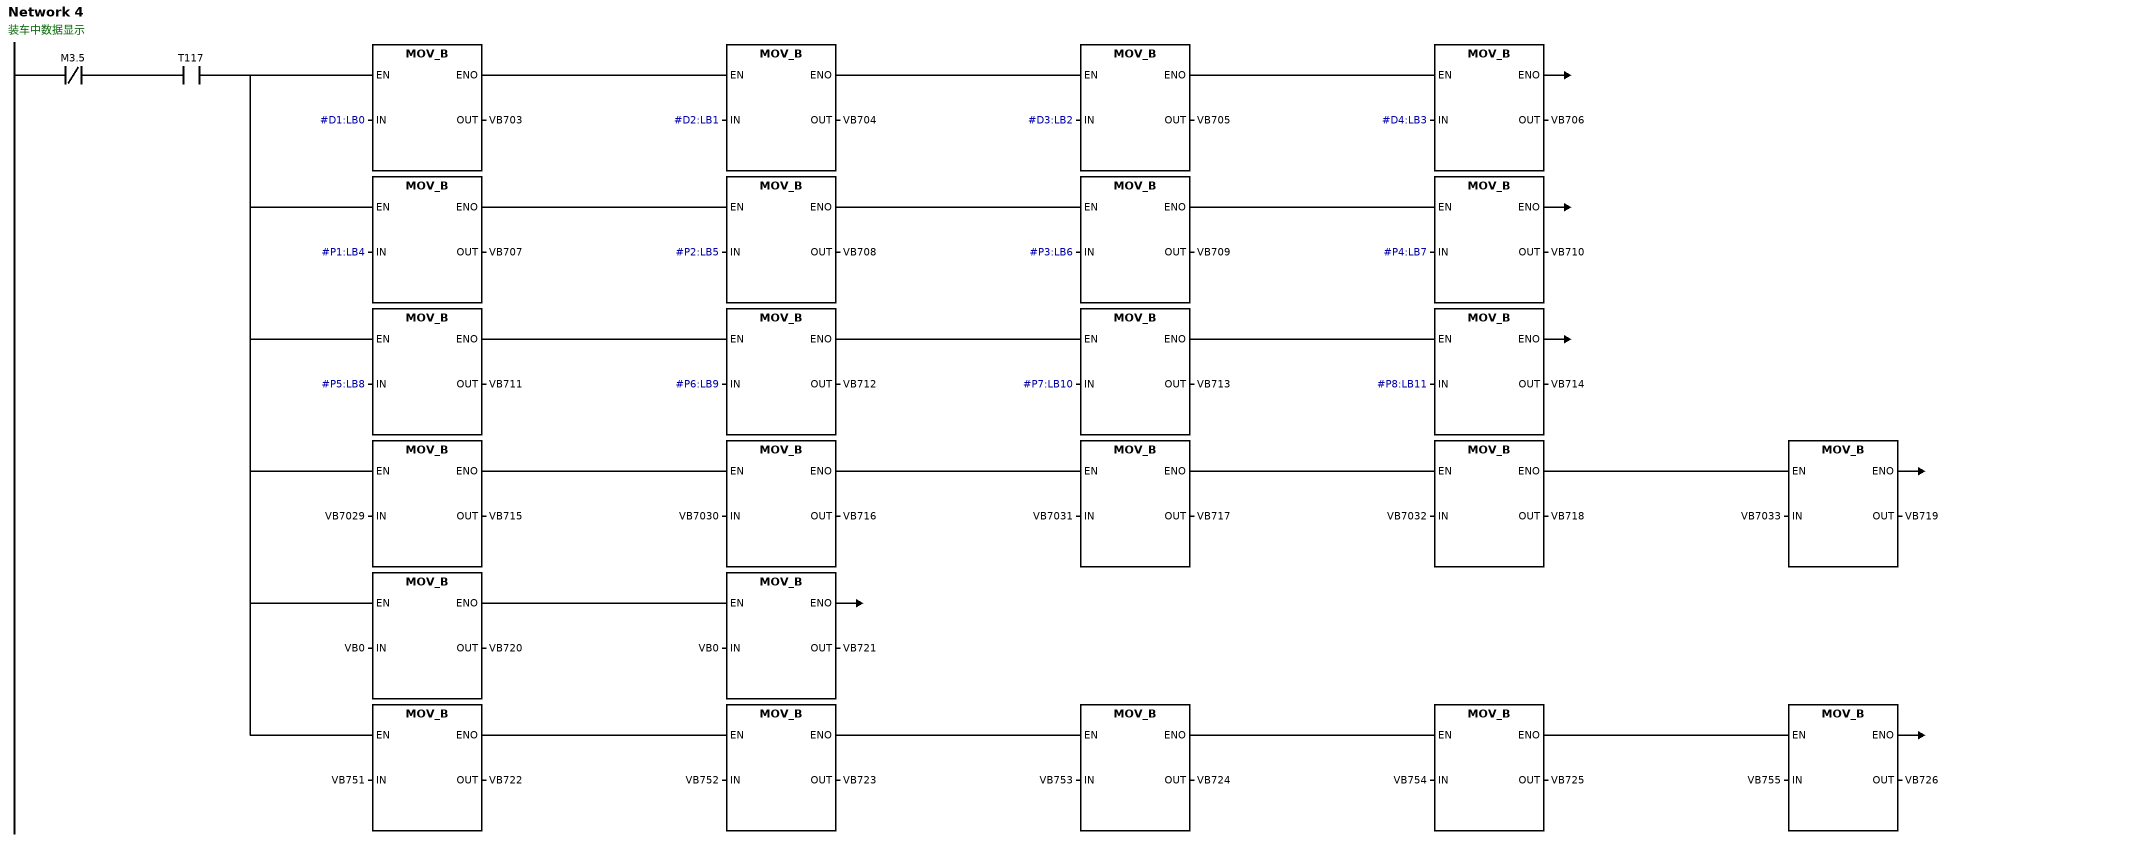
[picture p48: SBR17 networks 4-4]
Network 4
// 装车中数据显示
LDN    M3.5
A      T117
LPS
MOVB   #D1:LB0, VB703
AENO
MOVB   #D2:LB1, VB704
AENO
MOVB   #D3:LB2, VB705
AENO
MOVB   #D4:LB3, VB706
LRD
MOVB   #P1:LB4, VB707
AENO
MOVB   #P2:LB5, VB708
AENO
MOVB   #P3:LB6, VB709
AENO
MOVB   #P4:LB7, VB710
LRD
MOVB   #P5:LB8, VB711
AENO
MOVB   #P6:LB9, VB712
AENO
MOVB   #P7:LB10, VB713
AENO
MOVB   #P8:LB11, VB714
LRD
MOVB   VB7029, VB715
AENO
MOVB   VB7030, VB716
AENO
MOVB   VB7031, VB717
AENO
MOVB   VB7032, VB718
AENO
MOVB   VB7033, VB719
LRD
MOVB   VB0, VB720
AENO
MOVB   VB0, VB721
LPP
MOVB   VB751, VB722
AENO
MOVB   VB752, VB723
AENO
MOVB   VB753, VB724
AENO
MOVB   VB754, VB725
AENO
MOVB   VB755, VB726
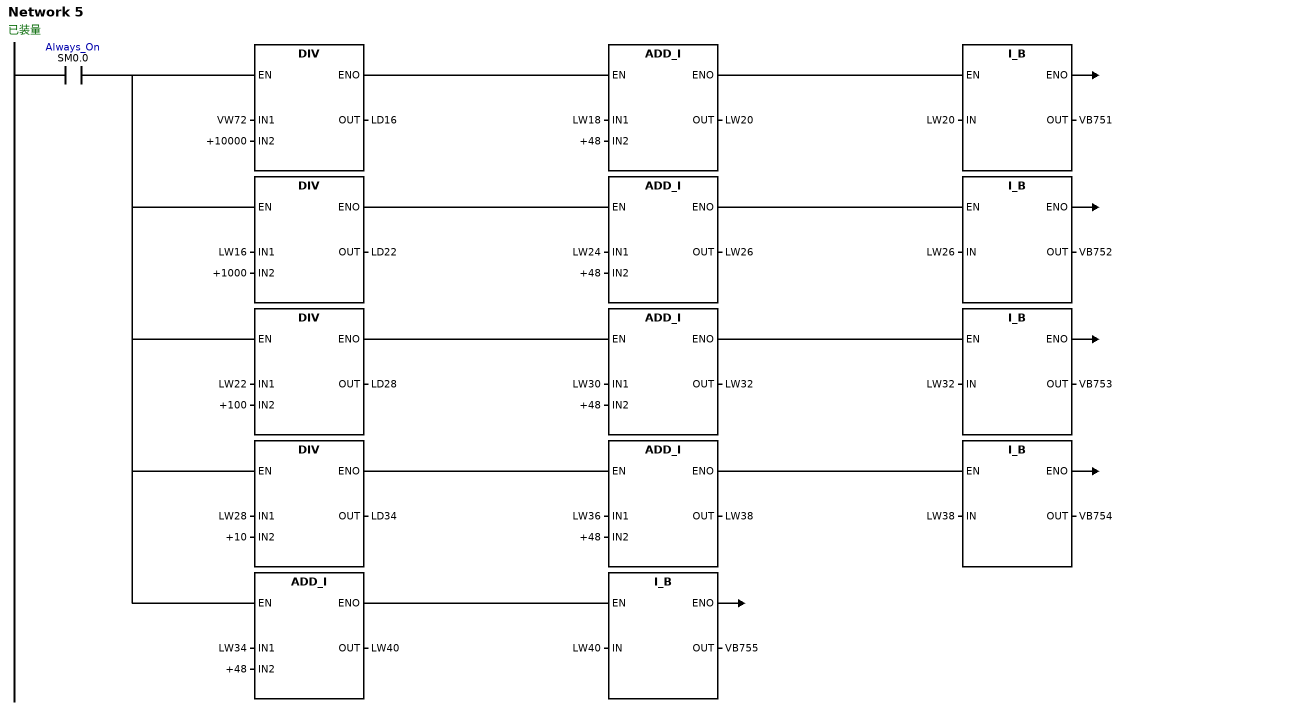
Network 5
// 已装量
LD     Always_On:SM0.0
LPS
MOVW   VW72, LW18
AENO
DIV    +10000, LD16
AENO
MOVW   LW18, LW20
AENO
+I     +48, LW20
AENO
ITB    LW20, VB751
LRD
MOVW   LW16, LW24
AENO
DIV    +1000, LD22
AENO
MOVW   LW24, LW26
AENO
+I     +48, LW26
AENO
ITB    LW26, VB752
LRD
MOVW   LW22, LW30
AENO
DIV    +100, LD28
AENO
MOVW   LW30, LW32
AENO
+I     +48, LW32
AENO
ITB    LW32, VB753
LRD
MOVW   LW28, LW36
AENO
DIV    +10, LD34
AENO
MOVW   LW36, LW38
AENO
+I     +48, LW38
AENO
ITB    LW38, VB754
LPP
MOVW   LW34, LW40
AENO
+I     +48, LW40
AENO
ITB    LW40, VB755
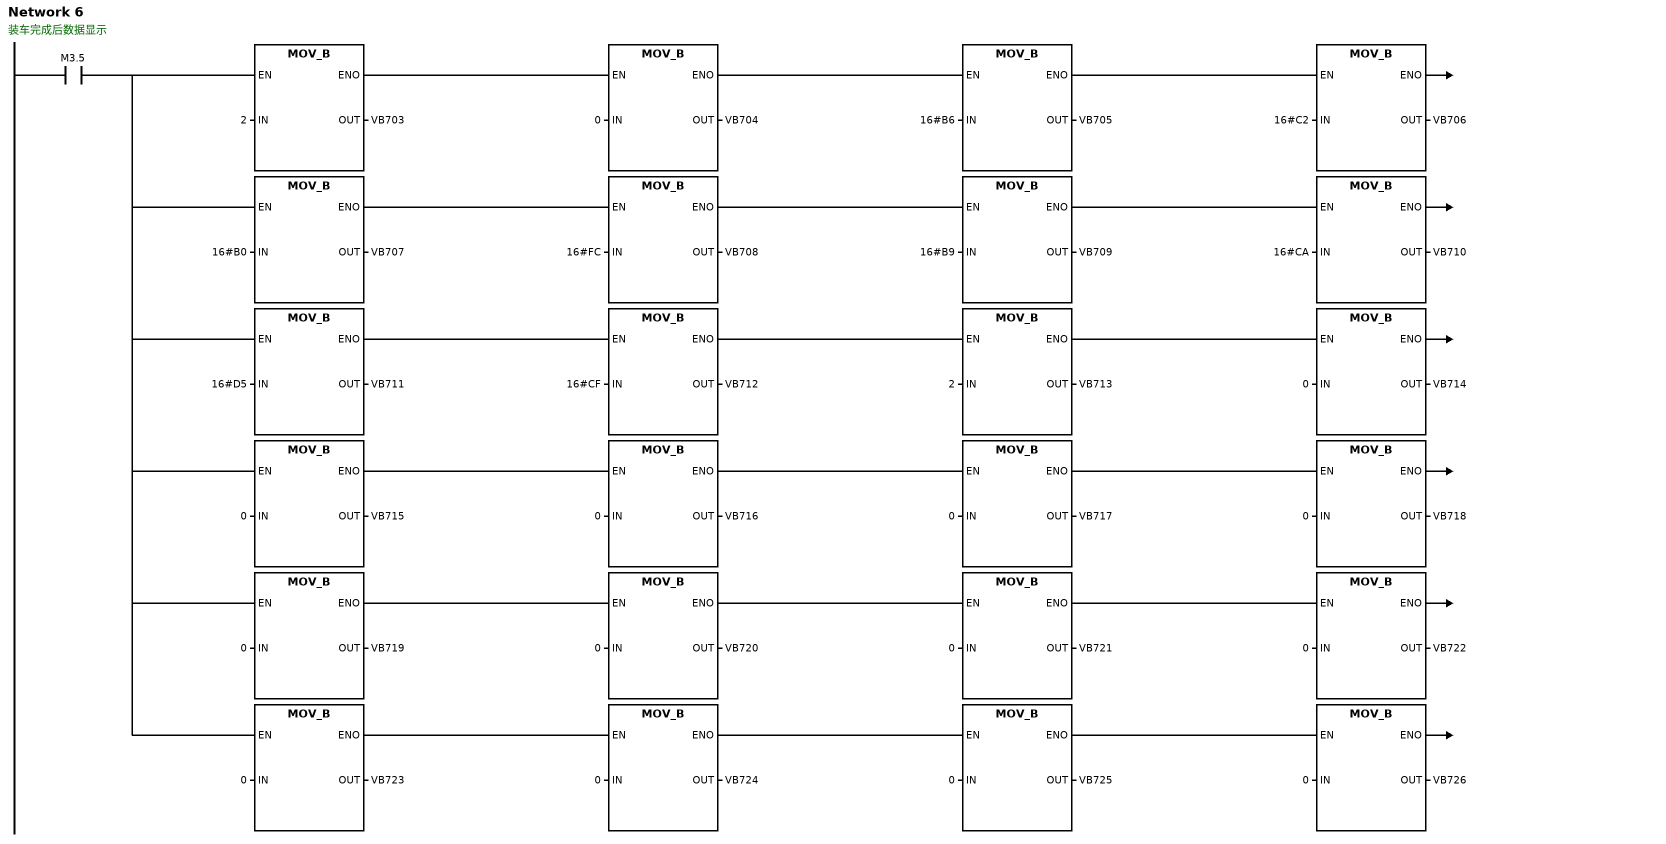
Network 6
// 装车完成后数据显示
LD     M3.5
LPS
MOVB   2, VB703
AENO
MOVB   0, VB704
AENO
MOVB   16#B6, VB705
AENO
MOVB   16#C2, VB706
LRD
MOVB   16#B0, VB707
AENO
MOVB   16#FC, VB708
AENO
MOVB   16#B9, VB709
AENO
MOVB   16#CA, VB710
LRD
MOVB   16#D5, VB711
AENO
MOVB   16#CF, VB712
AENO
MOVB   2, VB713
AENO
MOVB   0, VB714
LRD
MOVB   0, VB715
AENO
MOVB   0, VB716
AENO
MOVB   0, VB717
AENO
MOVB   0, VB718
LRD
MOVB   0, VB719
AENO
MOVB   0, VB720
AENO
MOVB   0, VB721
AENO
MOVB   0, VB722
LPP
MOVB   0, VB723
AENO
MOVB   0, VB724
AENO
MOVB   0, VB725
AENO
MOVB   0, VB726
END_SUBROUTINE_BLOCK

SUBROUTINE_BLOCK LED8:SBR18
TITLE=
VAR_INPUT
D1:BYTE;	// LB0 
D2:BYTE;	// LB1 
D3:BYTE;	// LB2 
D4:BYTE;	// LB3 
P1:BYTE;	// LB4 
P2:BYTE;	// LB5 
P3:BYTE;	// LB6 
P4:BYTE;	// LB7 
P5:BYTE;	// LB8 
P6:BYTE;	// LB9 
P7:BYTE;	// LB10 
P8:BYTE;	// LB11 
RUN:WORD;	// LW12 
END_VAR
BEGIN
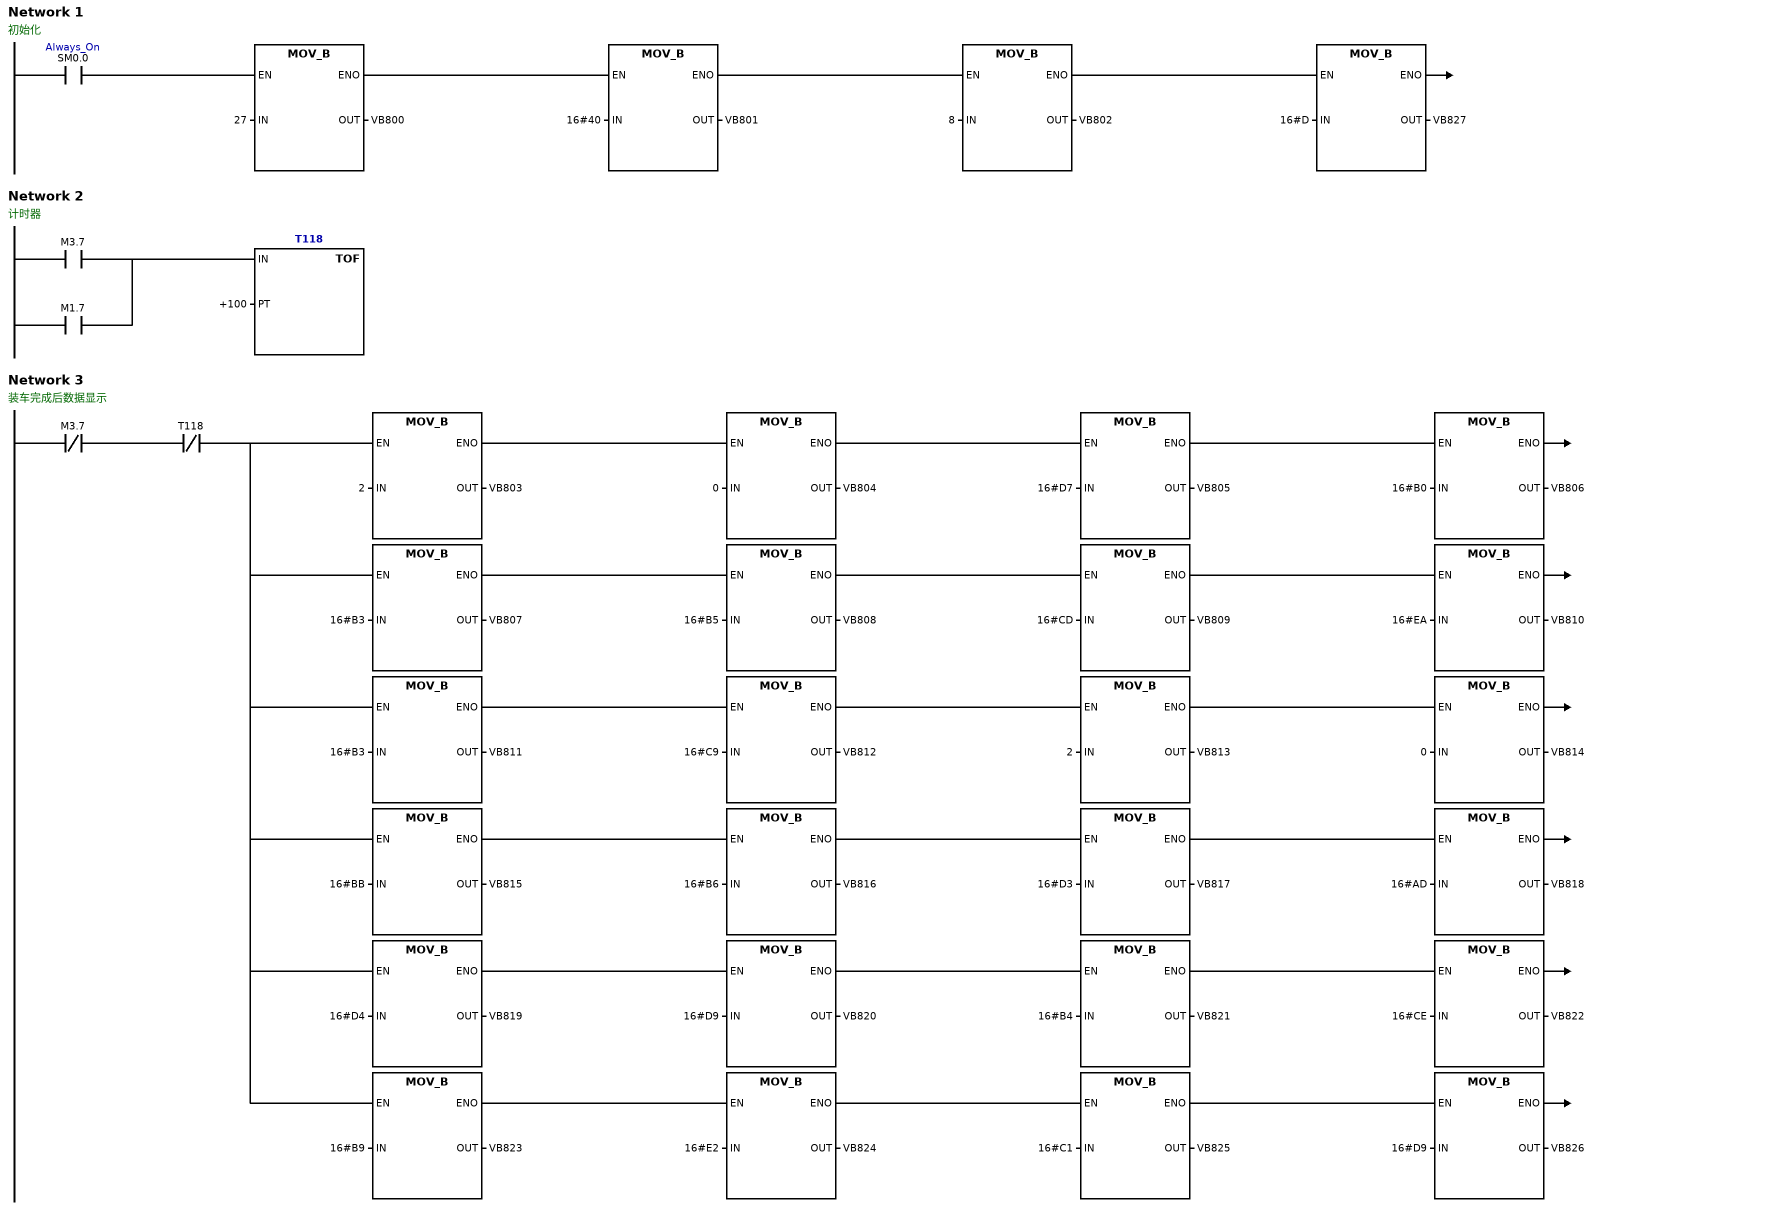
Network 1
// 初始化
LD     Always_On:SM0.0
MOVB   27, VB800
AENO
MOVB   16#40, VB801
AENO
MOVB   8, VB802
AENO
MOVB   16#D, VB827
Network 2
// 计时器
LD     M3.7
O      M1.7
TOF    T118, +100
Network 3
// 装车完成后数据显示
LDN    M3.7
AN     T118
LPS
MOVB   2, VB803
AENO
MOVB   0, VB804
AENO
MOVB   16#D7, VB805
AENO
MOVB   16#B0, VB806
LRD
MOVB   16#B3, VB807
AENO
MOVB   16#B5, VB808
AENO
MOVB   16#CD, VB809
AENO
MOVB   16#EA, VB810
LRD
MOVB   16#B3, VB811
AENO
MOVB   16#C9, VB812
AENO
MOVB   2, VB813
AENO
MOVB   0, VB814
LRD
MOVB   16#BB, VB815
AENO
MOVB   16#B6, VB816
AENO
MOVB   16#D3, VB817
AENO
MOVB   16#AD, VB818
LRD
MOVB   16#D4, VB819
AENO
MOVB   16#D9, VB820
AENO
MOVB   16#B4, VB821
AENO
MOVB   16#CE, VB822
LPP
MOVB   16#B9, VB823
AENO
MOVB   16#E2, VB824
AENO
MOVB   16#C1, VB825
AENO
MOVB   16#D9, VB826
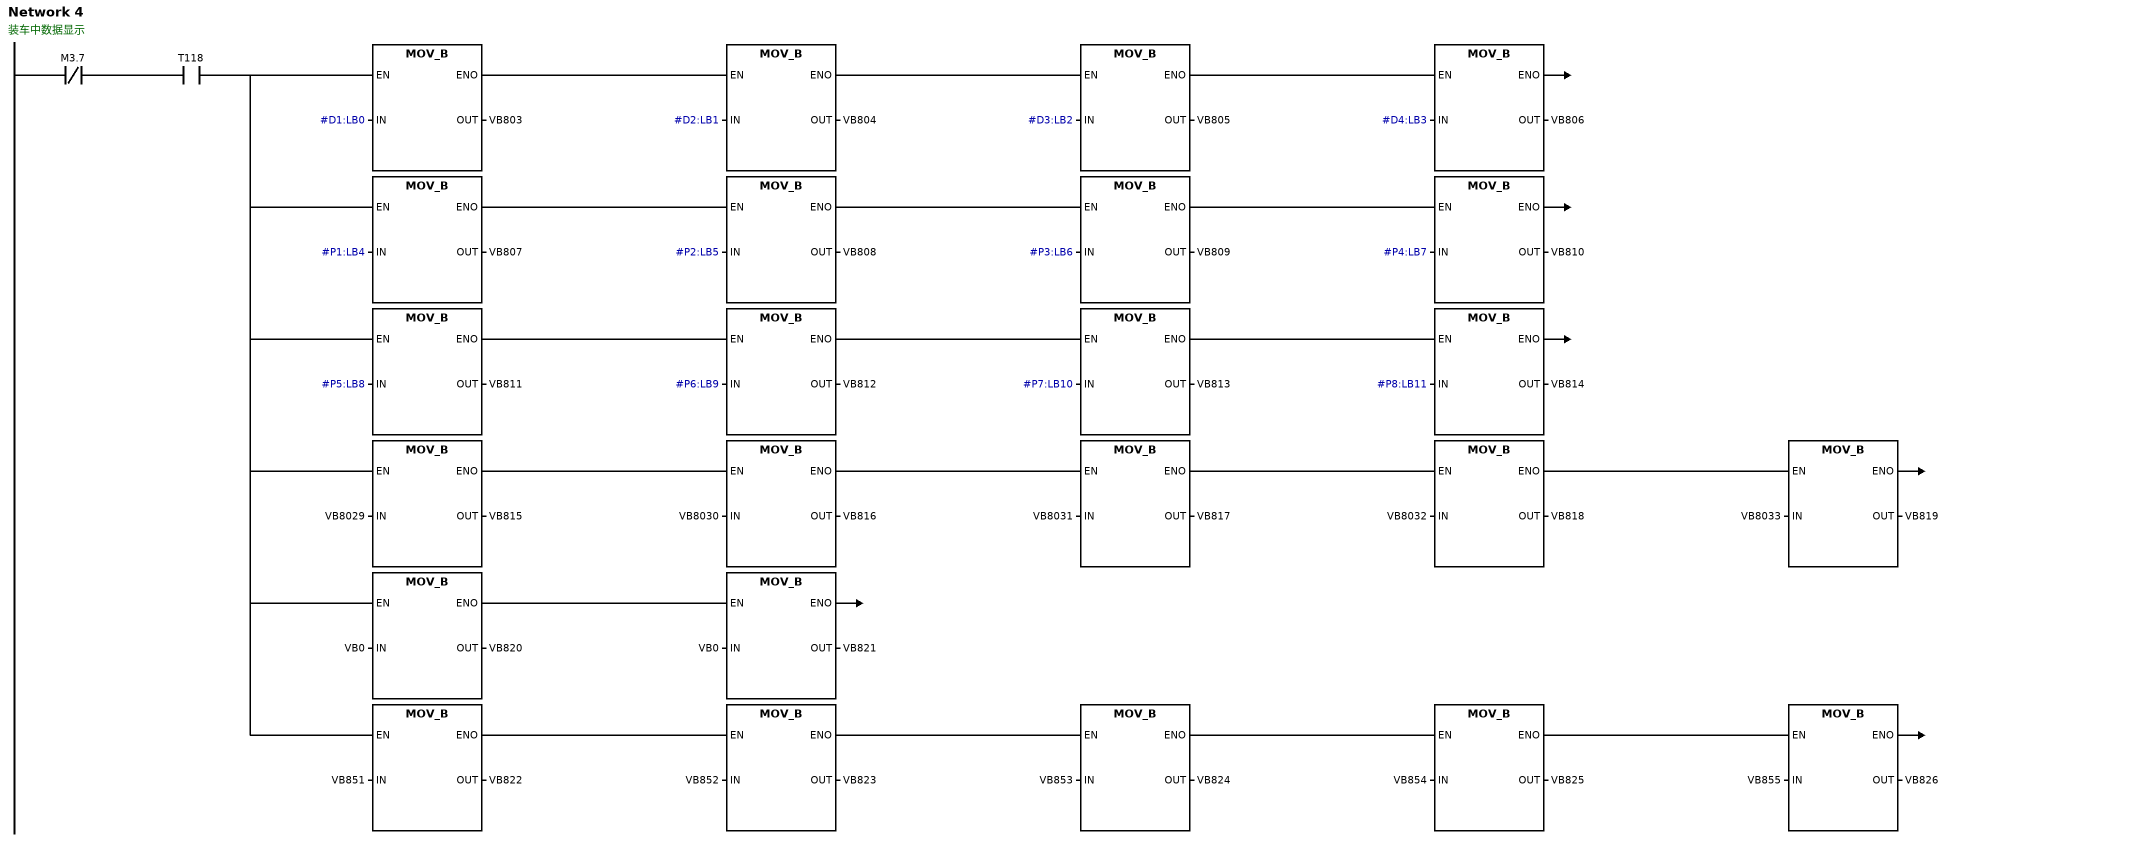
Network 4
// 装车中数据显示
LDN    M3.7
A      T118
LPS
MOVB   #D1:LB0, VB803
AENO
MOVB   #D2:LB1, VB804
AENO
MOVB   #D3:LB2, VB805
AENO
MOVB   #D4:LB3, VB806
LRD
MOVB   #P1:LB4, VB807
AENO
MOVB   #P2:LB5, VB808
AENO
MOVB   #P3:LB6, VB809
AENO
MOVB   #P4:LB7, VB810
LRD
MOVB   #P5:LB8, VB811
AENO
MOVB   #P6:LB9, VB812
AENO
MOVB   #P7:LB10, VB813
AENO
MOVB   #P8:LB11, VB814
LRD
MOVB   VB8029, VB815
AENO
MOVB   VB8030, VB816
AENO
MOVB   VB8031, VB817
AENO
MOVB   VB8032, VB818
AENO
MOVB   VB8033, VB819
LRD
MOVB   VB0, VB820
AENO
MOVB   VB0, VB821
LPP
MOVB   VB851, VB822
AENO
MOVB   VB852, VB823
AENO
MOVB   VB853, VB824
AENO
MOVB   VB854, VB825
AENO
MOVB   VB855, VB826
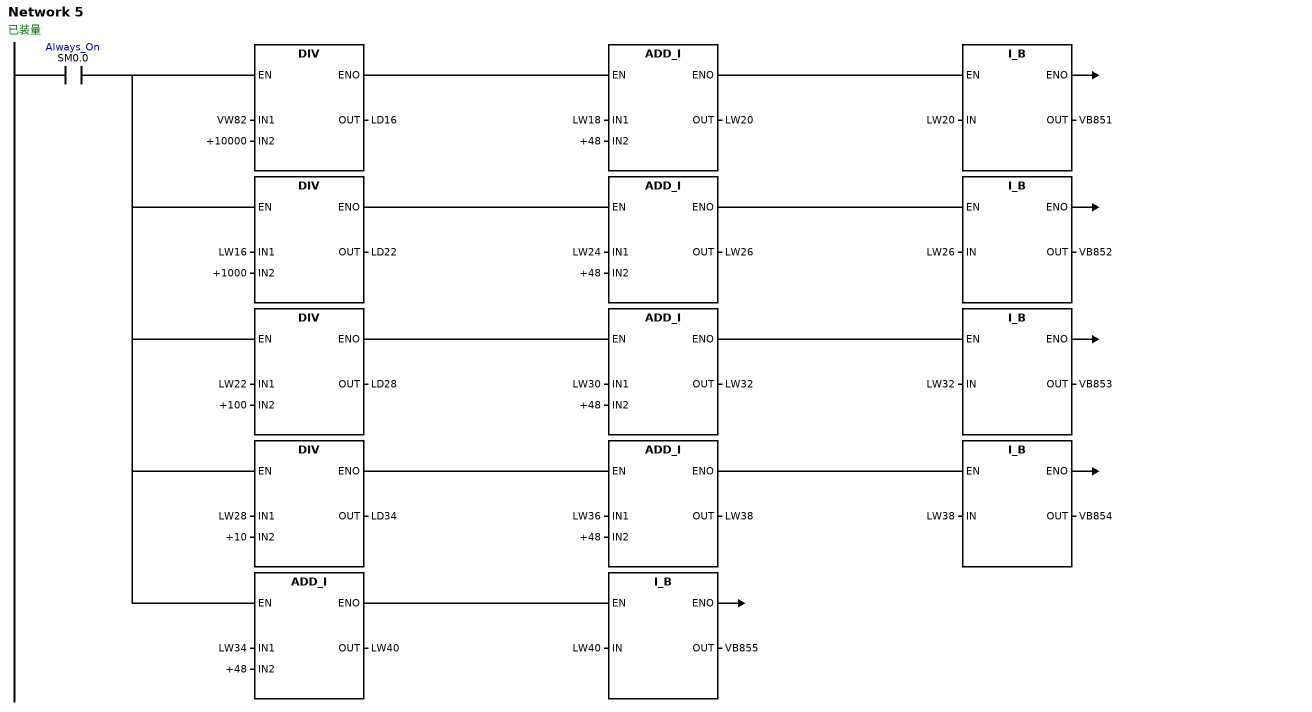
Network 5
// 已装量
LD     Always_On:SM0.0
LPS
MOVW   VW82, LW18
AENO
DIV    +10000, LD16
AENO
MOVW   LW18, LW20
AENO
+I     +48, LW20
AENO
ITB    LW20, VB851
LRD
MOVW   LW16, LW24
AENO
DIV    +1000, LD22
AENO
MOVW   LW24, LW26
AENO
+I     +48, LW26
AENO
ITB    LW26, VB852
LRD
MOVW   LW22, LW30
AENO
DIV    +100, LD28
AENO
MOVW   LW30, LW32
AENO
+I     +48, LW32
AENO
ITB    LW32, VB853
LRD
MOVW   LW28, LW36
AENO
DIV    +10, LD34
AENO
MOVW   LW36, LW38
AENO
+I     +48, LW38
AENO
ITB    LW38, VB854
LPP
MOVW   LW34, LW40
AENO
+I     +48, LW40
AENO
ITB    LW40, VB855
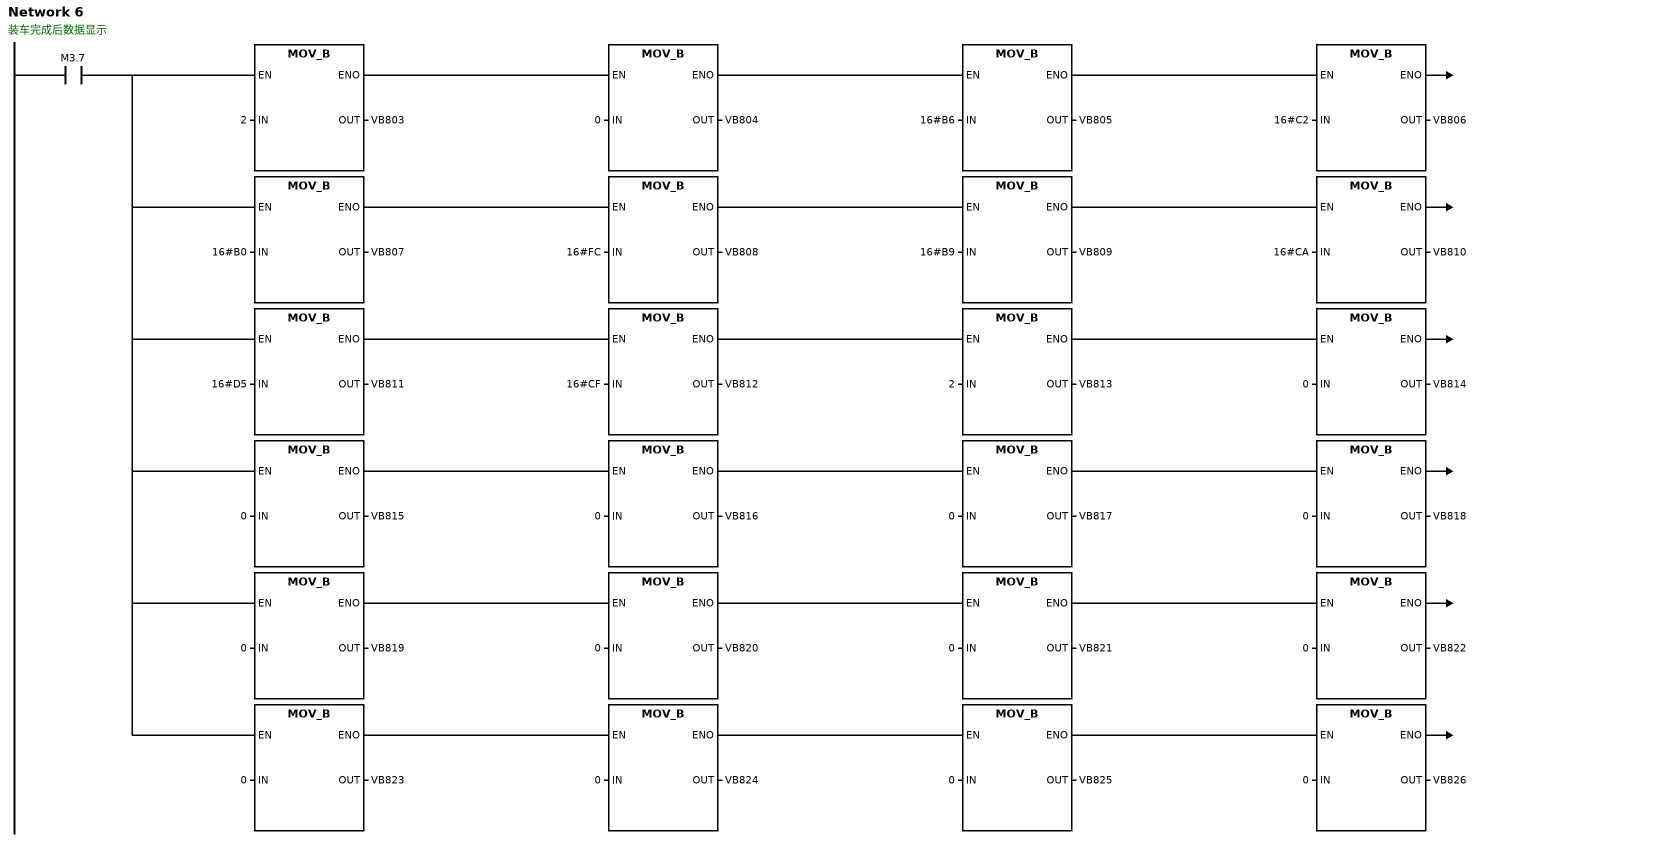
Network 6
// 装车完成后数据显示
LD     M3.7
LPS
MOVB   2, VB803
AENO
MOVB   0, VB804
AENO
MOVB   16#B6, VB805
AENO
MOVB   16#C2, VB806
LRD
MOVB   16#B0, VB807
AENO
MOVB   16#FC, VB808
AENO
MOVB   16#B9, VB809
AENO
MOVB   16#CA, VB810
LRD
MOVB   16#D5, VB811
AENO
MOVB   16#CF, VB812
AENO
MOVB   2, VB813
AENO
MOVB   0, VB814
LRD
MOVB   0, VB815
AENO
MOVB   0, VB816
AENO
MOVB   0, VB817
AENO
MOVB   0, VB818
LRD
MOVB   0, VB819
AENO
MOVB   0, VB820
AENO
MOVB   0, VB821
AENO
MOVB   0, VB822
LPP
MOVB   0, VB823
AENO
MOVB   0, VB824
AENO
MOVB   0, VB825
AENO
MOVB   0, VB826
END_SUBROUTINE_BLOCK

// SBR19: protected block, not included

// SBR20: protected block, not included

SUBROUTINE_BLOCK N1收:SBR21
TITLE=
VAR_OUTPUT
总袋数1:WORD;	// LW0 
袋长1:WORD;	// LW2 
END_VAR
VAR
TEMP1:WORD;	// LW4 
TEMP2:WORD;	// LW6 
TEMP3:WORD;	// LW8 
TEMP4:WORD;	// LW10 
TEMP5:WORD;	// LW12 
TEMP6:WORD;	// LW14 
TEMP7:WORD;	// LW16 
TEMP8:WORD;	// LW18 
TEMP9:WORD;	// LW20 
TEMP10:WORD;	// LW22 
TEMP11:WORD;	// LW24 
TEMP12:WORD;	// LW26 
TEMP13:WORD;	// LW28 
TEMP14:WORD;	// LW30 
TEMP15:WORD;	// LW32 
TEMP16:WORD;	// LW34 
TEMP17:WORD;	// LW36 
TEMP18:WORD;	// LW38 
TEMP19:WORD;	// LW40 
TEMP20:WORD;	// LW42 
TEMP21:WORD;	// LW44 
END_VAR
BEGIN
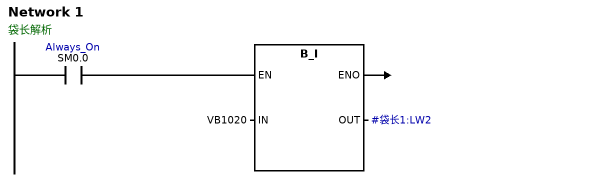
Network 1
// 袋长解析
LD     Always_On:SM0.0
BTI    VB1020, #袋长1:LW2
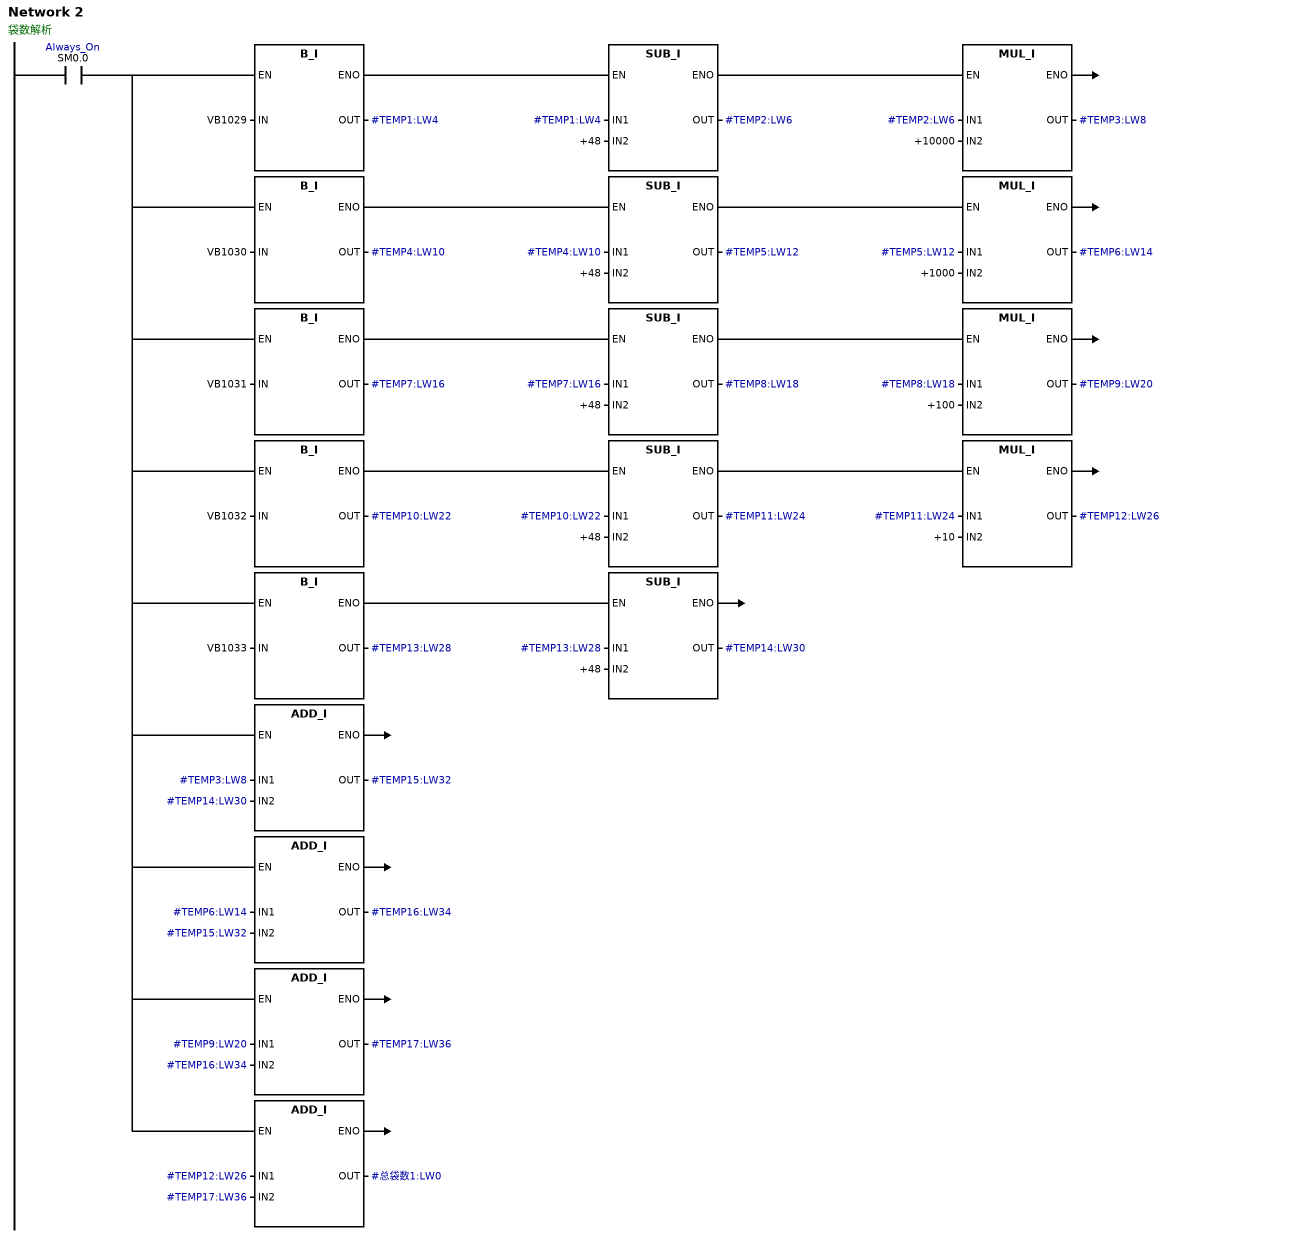
Network 2
// 袋数解析
LD     Always_On:SM0.0
LPS
BTI    VB1029, #TEMP1:LW4
AENO
MOVW   #TEMP1:LW4, #TEMP2:LW6
AENO
-I     +48, #TEMP2:LW6
AENO
MOVW   #TEMP2:LW6, #TEMP3:LW8
*I     +10000, #TEMP3:LW8
LRD
BTI    VB1030, #TEMP4:LW10
AENO
MOVW   #TEMP4:LW10, #TEMP5:LW12
AENO
-I     +48, #TEMP5:LW12
AENO
MOVW   #TEMP5:LW12, #TEMP6:LW14
*I     +1000, #TEMP6:LW14
LRD
BTI    VB1031, #TEMP7:LW16
AENO
MOVW   #TEMP7:LW16, #TEMP8:LW18
AENO
-I     +48, #TEMP8:LW18
AENO
MOVW   #TEMP8:LW18, #TEMP9:LW20
*I     +100, #TEMP9:LW20
LRD
BTI    VB1032, #TEMP10:LW22
AENO
MOVW   #TEMP10:LW22, #TEMP11:LW24
AENO
-I     +48, #TEMP11:LW24
AENO
MOVW   #TEMP11:LW24, #TEMP12:LW26
*I     +10, #TEMP12:LW26
LRD
BTI    VB1033, #TEMP13:LW28
AENO
MOVW   #TEMP13:LW28, #TEMP14:LW30
-I     +48, #TEMP14:LW30
LRD
MOVW   #TEMP3:LW8, #TEMP15:LW32
+I     #TEMP14:LW30, #TEMP15:LW32
LRD
MOVW   #TEMP6:LW14, #TEMP16:LW34
+I     #TEMP15:LW32, #TEMP16:LW34
LRD
MOVW   #TEMP9:LW20, #TEMP17:LW36
+I     #TEMP16:LW34, #TEMP17:LW36
LPP
MOVW   #TEMP12:LW26, #总袋数1:LW0
+I     #TEMP17:LW36, #总袋数1:LW0
END_SUBROUTINE_BLOCK

SUBROUTINE_BLOCK N2收:SBR22
TITLE=
VAR_OUTPUT
总袋数1:WORD;	// LW0 
袋长1:WORD;	// LW2 
END_VAR
VAR
TEMP1:WORD;	// LW4 
TEMP2:WORD;	// LW6 
TEMP3:WORD;	// LW8 
TEMP4:WORD;	// LW10 
TEMP5:WORD;	// LW12 
TEMP6:WORD;	// LW14 
TEMP7:WORD;	// LW16 
TEMP8:WORD;	// LW18 
TEMP9:WORD;	// LW20 
TEMP10:WORD;	// LW22 
TEMP11:WORD;	// LW24 
TEMP12:WORD;	// LW26 
TEMP13:WORD;	// LW28 
TEMP14:WORD;	// LW30 
TEMP15:WORD;	// LW32 
TEMP16:WORD;	// LW34 
TEMP17:WORD;	// LW36 
TEMP18:WORD;	// LW38 
TEMP19:WORD;	// LW40 
TEMP20:WORD;	// LW42 
TEMP21:WORD;	// LW44 
END_VAR
BEGIN
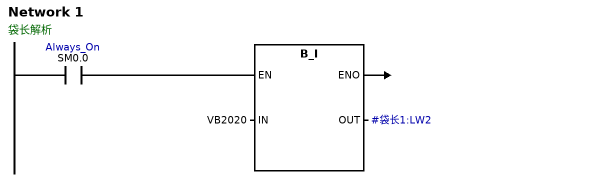
Network 1
// 袋长解析
LD     Always_On:SM0.0
BTI    VB2020, #袋长1:LW2
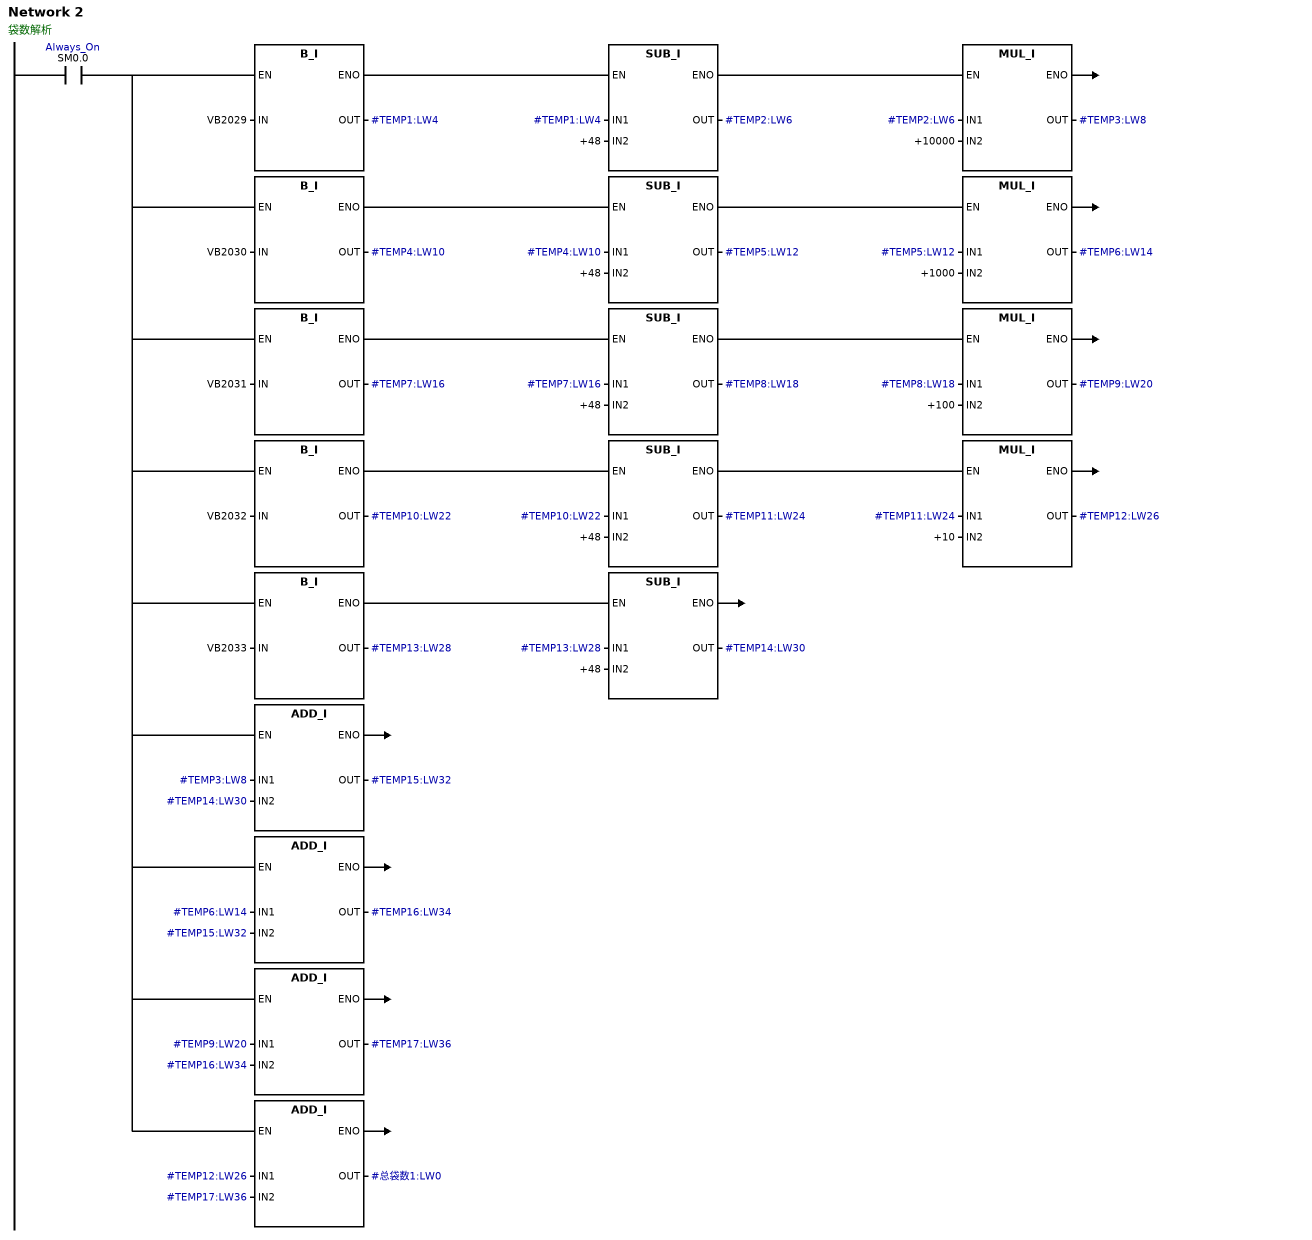
Network 2
// 袋数解析
LD     Always_On:SM0.0
LPS
BTI    VB2029, #TEMP1:LW4
AENO
MOVW   #TEMP1:LW4, #TEMP2:LW6
AENO
-I     +48, #TEMP2:LW6
AENO
MOVW   #TEMP2:LW6, #TEMP3:LW8
*I     +10000, #TEMP3:LW8
LRD
BTI    VB2030, #TEMP4:LW10
AENO
MOVW   #TEMP4:LW10, #TEMP5:LW12
AENO
-I     +48, #TEMP5:LW12
AENO
MOVW   #TEMP5:LW12, #TEMP6:LW14
*I     +1000, #TEMP6:LW14
LRD
BTI    VB2031, #TEMP7:LW16
AENO
MOVW   #TEMP7:LW16, #TEMP8:LW18
AENO
-I     +48, #TEMP8:LW18
AENO
MOVW   #TEMP8:LW18, #TEMP9:LW20
*I     +100, #TEMP9:LW20
LRD
BTI    VB2032, #TEMP10:LW22
AENO
MOVW   #TEMP10:LW22, #TEMP11:LW24
AENO
-I     +48, #TEMP11:LW24
AENO
MOVW   #TEMP11:LW24, #TEMP12:LW26
*I     +10, #TEMP12:LW26
LRD
BTI    VB2033, #TEMP13:LW28
AENO
MOVW   #TEMP13:LW28, #TEMP14:LW30
-I     +48, #TEMP14:LW30
LRD
MOVW   #TEMP3:LW8, #TEMP15:LW32
+I     #TEMP14:LW30, #TEMP15:LW32
LRD
MOVW   #TEMP6:LW14, #TEMP16:LW34
+I     #TEMP15:LW32, #TEMP16:LW34
LRD
MOVW   #TEMP9:LW20, #TEMP17:LW36
+I     #TEMP16:LW34, #TEMP17:LW36
LPP
MOVW   #TEMP12:LW26, #总袋数1:LW0
+I     #TEMP17:LW36, #总袋数1:LW0
END_SUBROUTINE_BLOCK

SUBROUTINE_BLOCK N3收:SBR23
TITLE=
VAR_OUTPUT
总袋数1:WORD;	// LW0 
袋长1:WORD;	// LW2 
END_VAR
VAR
TEMP1:WORD;	// LW4 
TEMP2:WORD;	// LW6 
TEMP3:WORD;	// LW8 
TEMP4:WORD;	// LW10 
TEMP5:WORD;	// LW12 
TEMP6:WORD;	// LW14 
TEMP7:WORD;	// LW16 
TEMP8:WORD;	// LW18 
TEMP9:WORD;	// LW20 
TEMP10:WORD;	// LW22 
TEMP11:WORD;	// LW24 
TEMP12:WORD;	// LW26 
TEMP13:WORD;	// LW28 
TEMP14:WORD;	// LW30 
TEMP15:WORD;	// LW32 
TEMP16:WORD;	// LW34 
TEMP17:WORD;	// LW36 
TEMP18:WORD;	// LW38 
TEMP19:WORD;	// LW40 
TEMP20:WORD;	// LW42 
TEMP21:WORD;	// LW44 
END_VAR
BEGIN
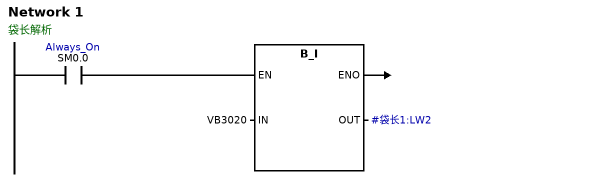
Network 1
// 袋长解析
LD     Always_On:SM0.0
BTI    VB3020, #袋长1:LW2
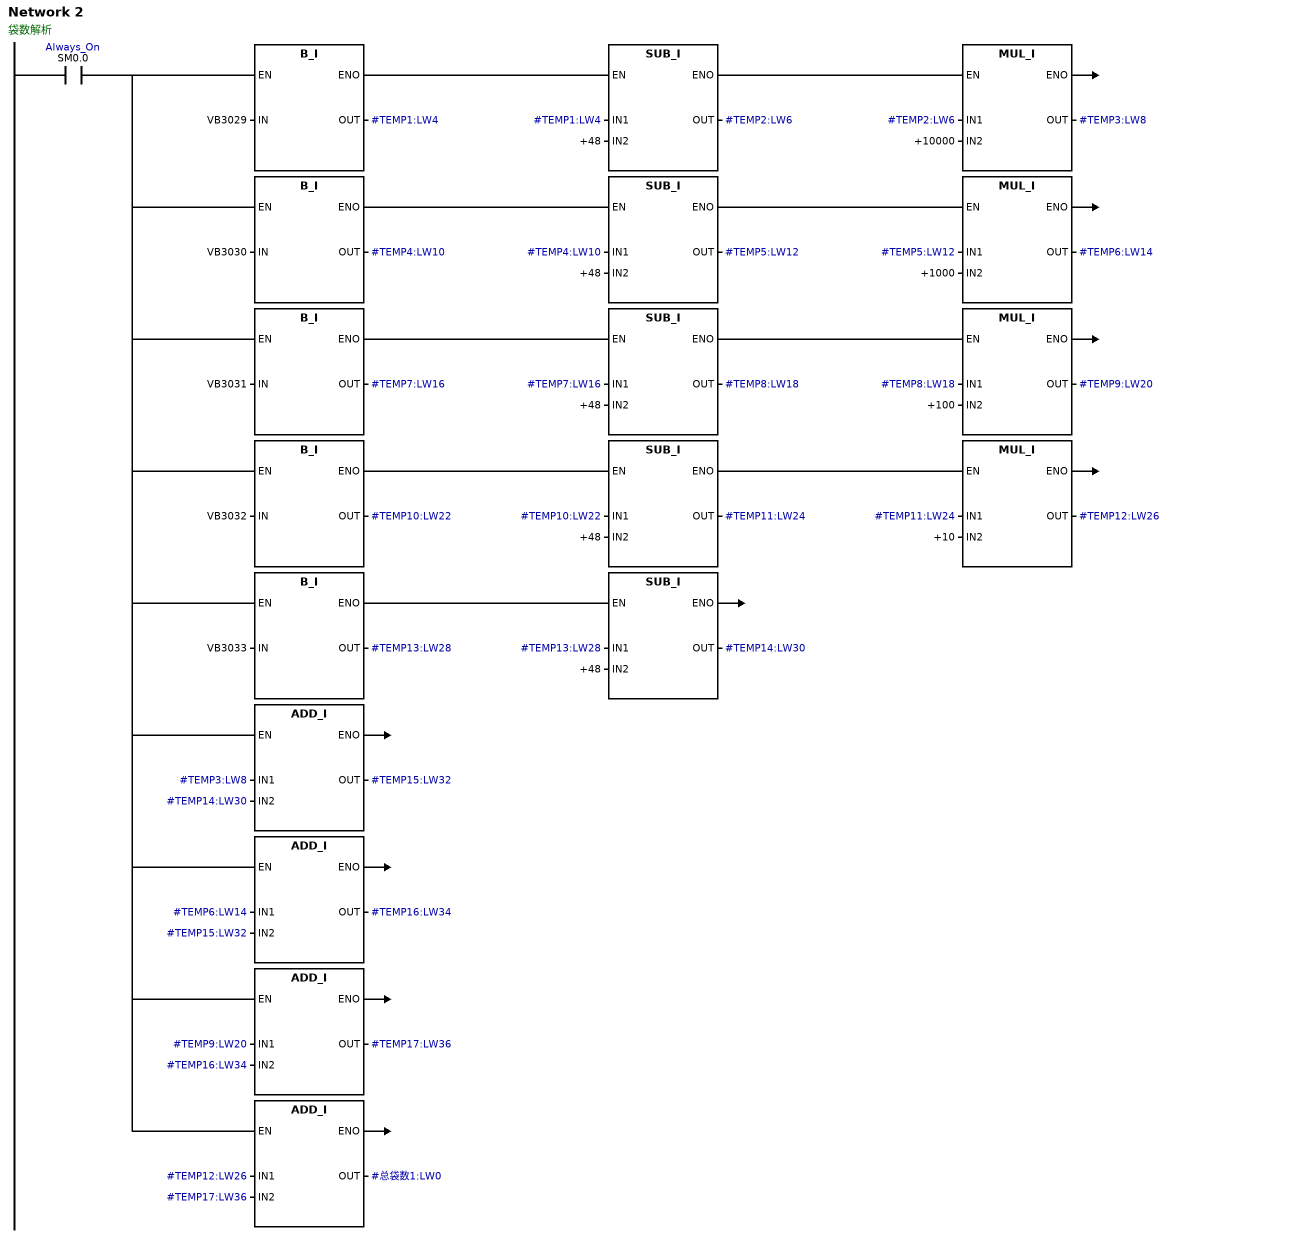
Network 2
// 袋数解析
LD     Always_On:SM0.0
LPS
BTI    VB3029, #TEMP1:LW4
AENO
MOVW   #TEMP1:LW4, #TEMP2:LW6
AENO
-I     +48, #TEMP2:LW6
AENO
MOVW   #TEMP2:LW6, #TEMP3:LW8
*I     +10000, #TEMP3:LW8
LRD
BTI    VB3030, #TEMP4:LW10
AENO
MOVW   #TEMP4:LW10, #TEMP5:LW12
AENO
-I     +48, #TEMP5:LW12
AENO
MOVW   #TEMP5:LW12, #TEMP6:LW14
*I     +1000, #TEMP6:LW14
LRD
BTI    VB3031, #TEMP7:LW16
AENO
MOVW   #TEMP7:LW16, #TEMP8:LW18
AENO
-I     +48, #TEMP8:LW18
AENO
MOVW   #TEMP8:LW18, #TEMP9:LW20
*I     +100, #TEMP9:LW20
LRD
BTI    VB3032, #TEMP10:LW22
AENO
MOVW   #TEMP10:LW22, #TEMP11:LW24
AENO
-I     +48, #TEMP11:LW24
AENO
MOVW   #TEMP11:LW24, #TEMP12:LW26
*I     +10, #TEMP12:LW26
LRD
BTI    VB3033, #TEMP13:LW28
AENO
MOVW   #TEMP13:LW28, #TEMP14:LW30
-I     +48, #TEMP14:LW30
LRD
MOVW   #TEMP3:LW8, #TEMP15:LW32
+I     #TEMP14:LW30, #TEMP15:LW32
LRD
MOVW   #TEMP6:LW14, #TEMP16:LW34
+I     #TEMP15:LW32, #TEMP16:LW34
LRD
MOVW   #TEMP9:LW20, #TEMP17:LW36
+I     #TEMP16:LW34, #TEMP17:LW36
LPP
MOVW   #TEMP12:LW26, #总袋数1:LW0
+I     #TEMP17:LW36, #总袋数1:LW0
END_SUBROUTINE_BLOCK

SUBROUTINE_BLOCK N4收:SBR24
TITLE=
VAR_OUTPUT
总袋数1:WORD;	// LW0 
袋长1:WORD;	// LW2 
END_VAR
VAR
TEMP1:WORD;	// LW4 
TEMP2:WORD;	// LW6 
TEMP3:WORD;	// LW8 
TEMP4:WORD;	// LW10 
TEMP5:WORD;	// LW12 
TEMP6:WORD;	// LW14 
TEMP7:WORD;	// LW16 
TEMP8:WORD;	// LW18 
TEMP9:WORD;	// LW20 
TEMP10:WORD;	// LW22 
TEMP11:WORD;	// LW24 
TEMP12:WORD;	// LW26 
TEMP13:WORD;	// LW28 
TEMP14:WORD;	// LW30 
TEMP15:WORD;	// LW32 
TEMP16:WORD;	// LW34 
TEMP17:WORD;	// LW36 
TEMP18:WORD;	// LW38 
TEMP19:WORD;	// LW40 
TEMP20:WORD;	// LW42 
TEMP21:WORD;	// LW44 
END_VAR
BEGIN
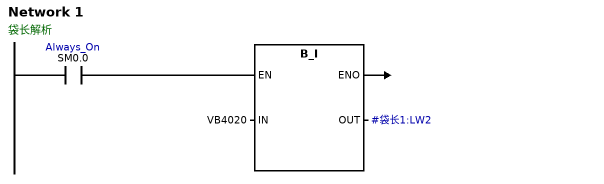
Network 1
// 袋长解析
LD     Always_On:SM0.0
BTI    VB4020, #袋长1:LW2
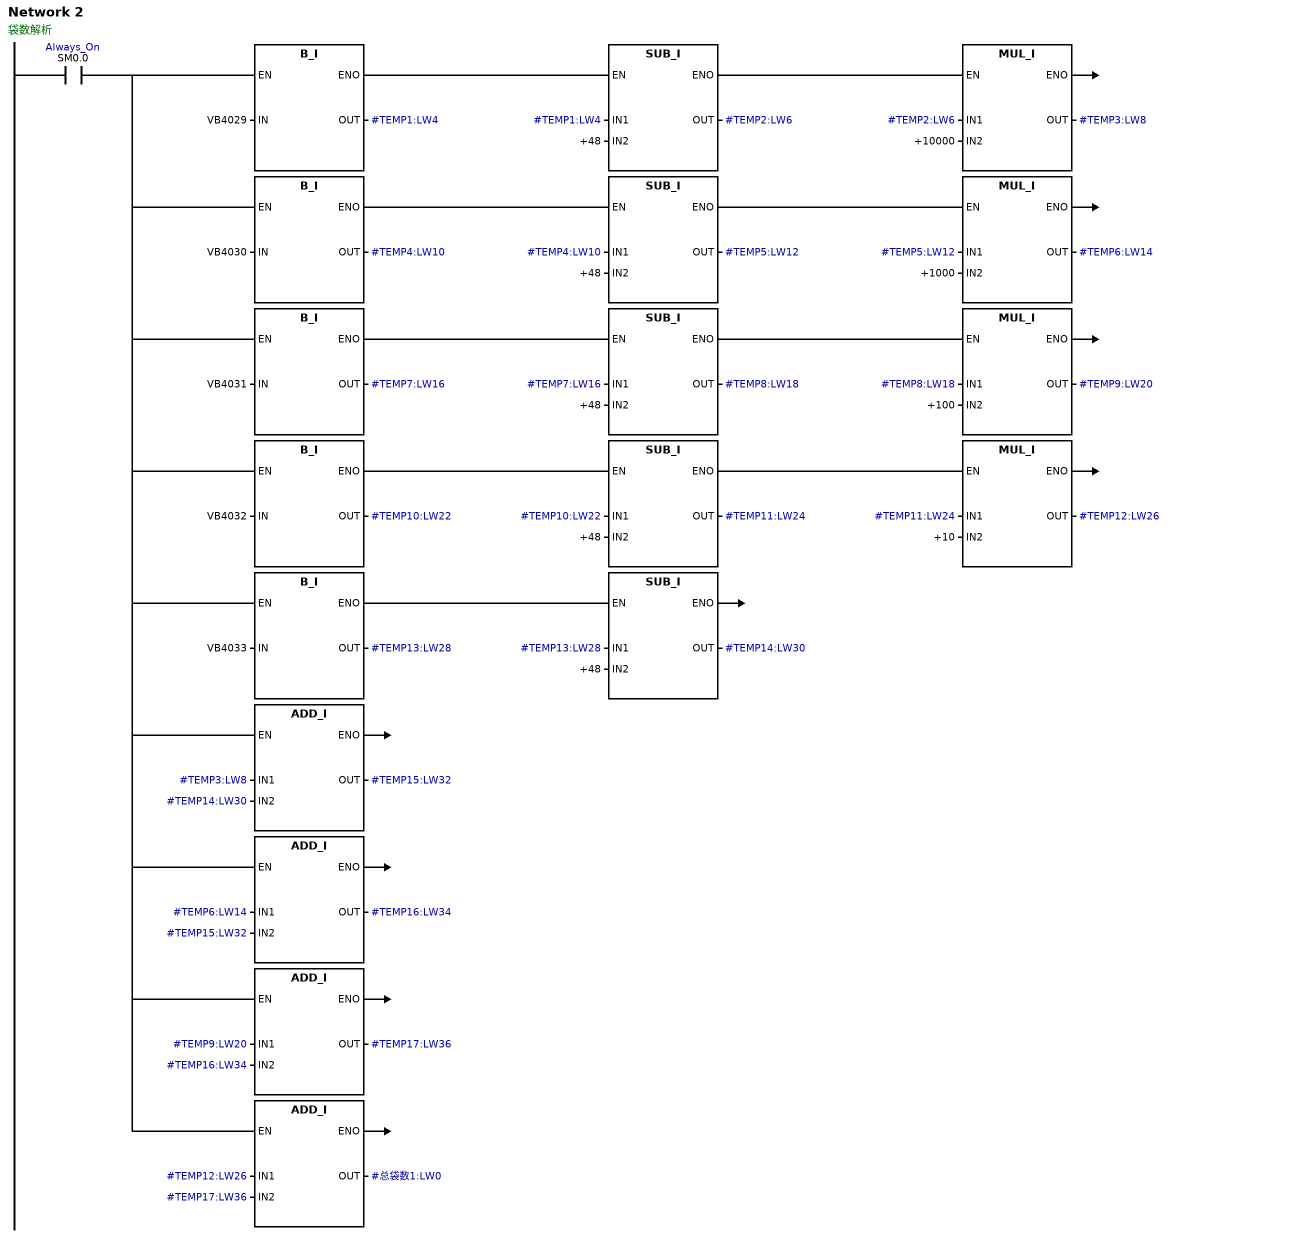
Network 2
// 袋数解析
LD     Always_On:SM0.0
LPS
BTI    VB4029, #TEMP1:LW4
AENO
MOVW   #TEMP1:LW4, #TEMP2:LW6
AENO
-I     +48, #TEMP2:LW6
AENO
MOVW   #TEMP2:LW6, #TEMP3:LW8
*I     +10000, #TEMP3:LW8
LRD
BTI    VB4030, #TEMP4:LW10
AENO
MOVW   #TEMP4:LW10, #TEMP5:LW12
AENO
-I     +48, #TEMP5:LW12
AENO
MOVW   #TEMP5:LW12, #TEMP6:LW14
*I     +1000, #TEMP6:LW14
LRD
BTI    VB4031, #TEMP7:LW16
AENO
MOVW   #TEMP7:LW16, #TEMP8:LW18
AENO
-I     +48, #TEMP8:LW18
AENO
MOVW   #TEMP8:LW18, #TEMP9:LW20
*I     +100, #TEMP9:LW20
LRD
BTI    VB4032, #TEMP10:LW22
AENO
MOVW   #TEMP10:LW22, #TEMP11:LW24
AENO
-I     +48, #TEMP11:LW24
AENO
MOVW   #TEMP11:LW24, #TEMP12:LW26
*I     +10, #TEMP12:LW26
LRD
BTI    VB4033, #TEMP13:LW28
AENO
MOVW   #TEMP13:LW28, #TEMP14:LW30
-I     +48, #TEMP14:LW30
LRD
MOVW   #TEMP3:LW8, #TEMP15:LW32
+I     #TEMP14:LW30, #TEMP15:LW32
LRD
MOVW   #TEMP6:LW14, #TEMP16:LW34
+I     #TEMP15:LW32, #TEMP16:LW34
LRD
MOVW   #TEMP9:LW20, #TEMP17:LW36
+I     #TEMP16:LW34, #TEMP17:LW36
LPP
MOVW   #TEMP12:LW26, #总袋数1:LW0
+I     #TEMP17:LW36, #总袋数1:LW0
END_SUBROUTINE_BLOCK

SUBROUTINE_BLOCK N5收:SBR25
TITLE=
VAR_OUTPUT
总袋数1:WORD;	// LW0 
袋长1:WORD;	// LW2 
END_VAR
VAR
TEMP1:WORD;	// LW4 
TEMP2:WORD;	// LW6 
TEMP3:WORD;	// LW8 
TEMP4:WORD;	// LW10 
TEMP5:WORD;	// LW12 
TEMP6:WORD;	// LW14 
TEMP7:WORD;	// LW16 
TEMP8:WORD;	// LW18 
TEMP9:WORD;	// LW20 
TEMP10:WORD;	// LW22 
TEMP11:WORD;	// LW24 
TEMP12:WORD;	// LW26 
TEMP13:WORD;	// LW28 
TEMP14:WORD;	// LW30 
TEMP15:WORD;	// LW32 
TEMP16:WORD;	// LW34 
TEMP17:WORD;	// LW36 
TEMP18:WORD;	// LW38 
TEMP19:WORD;	// LW40 
TEMP20:WORD;	// LW42 
TEMP21:WORD;	// LW44 
END_VAR
BEGIN
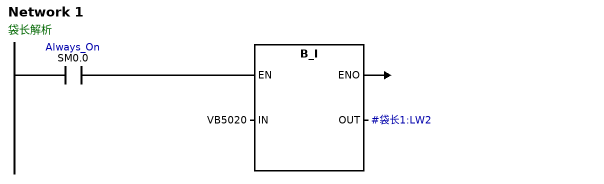
Network 1
// 袋长解析
LD     Always_On:SM0.0
BTI    VB5020, #袋长1:LW2
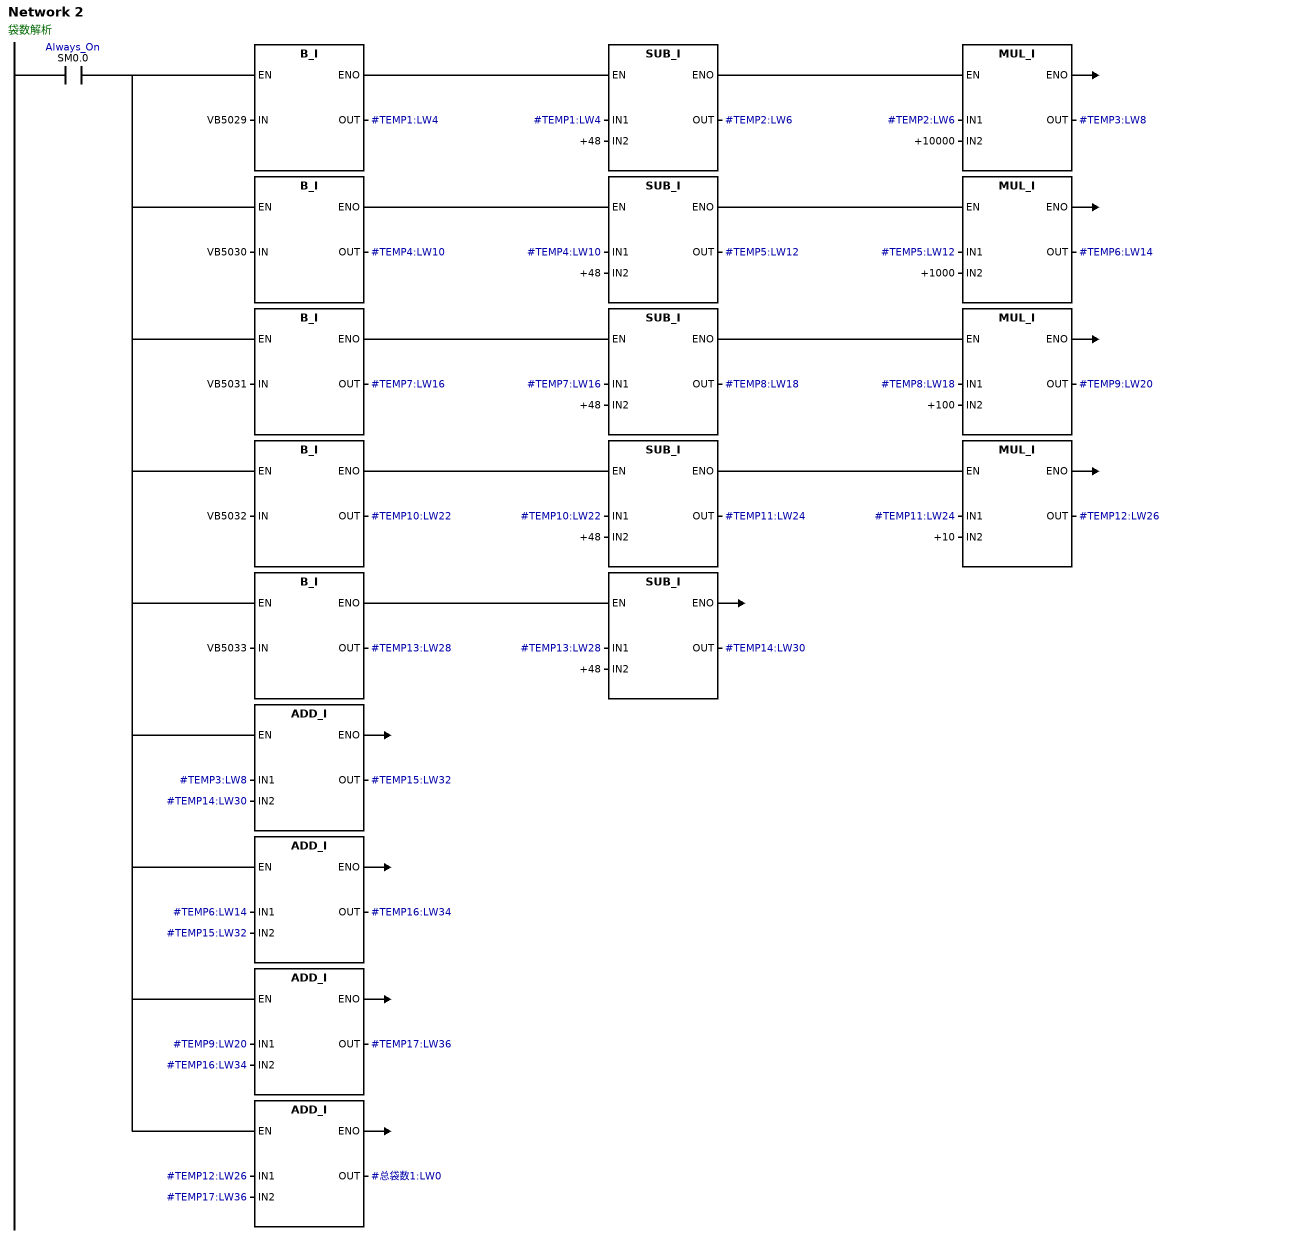
Network 2
// 袋数解析
LD     Always_On:SM0.0
LPS
BTI    VB5029, #TEMP1:LW4
AENO
MOVW   #TEMP1:LW4, #TEMP2:LW6
AENO
-I     +48, #TEMP2:LW6
AENO
MOVW   #TEMP2:LW6, #TEMP3:LW8
*I     +10000, #TEMP3:LW8
LRD
BTI    VB5030, #TEMP4:LW10
AENO
MOVW   #TEMP4:LW10, #TEMP5:LW12
AENO
-I     +48, #TEMP5:LW12
AENO
MOVW   #TEMP5:LW12, #TEMP6:LW14
*I     +1000, #TEMP6:LW14
LRD
BTI    VB5031, #TEMP7:LW16
AENO
MOVW   #TEMP7:LW16, #TEMP8:LW18
AENO
-I     +48, #TEMP8:LW18
AENO
MOVW   #TEMP8:LW18, #TEMP9:LW20
*I     +100, #TEMP9:LW20
LRD
BTI    VB5032, #TEMP10:LW22
AENO
MOVW   #TEMP10:LW22, #TEMP11:LW24
AENO
-I     +48, #TEMP11:LW24
AENO
MOVW   #TEMP11:LW24, #TEMP12:LW26
*I     +10, #TEMP12:LW26
LRD
BTI    VB5033, #TEMP13:LW28
AENO
MOVW   #TEMP13:LW28, #TEMP14:LW30
-I     +48, #TEMP14:LW30
LRD
MOVW   #TEMP3:LW8, #TEMP15:LW32
+I     #TEMP14:LW30, #TEMP15:LW32
LRD
MOVW   #TEMP6:LW14, #TEMP16:LW34
+I     #TEMP15:LW32, #TEMP16:LW34
LRD
MOVW   #TEMP9:LW20, #TEMP17:LW36
+I     #TEMP16:LW34, #TEMP17:LW36
LPP
MOVW   #TEMP12:LW26, #总袋数1:LW0
+I     #TEMP17:LW36, #总袋数1:LW0
END_SUBROUTINE_BLOCK

SUBROUTINE_BLOCK N6收:SBR26
TITLE=
VAR_OUTPUT
总袋数1:WORD;	// LW0 
袋长1:WORD;	// LW2 
END_VAR
VAR
TEMP1:WORD;	// LW4 
TEMP2:WORD;	// LW6 
TEMP3:WORD;	// LW8 
TEMP4:WORD;	// LW10 
TEMP5:WORD;	// LW12 
TEMP6:WORD;	// LW14 
TEMP7:WORD;	// LW16 
TEMP8:WORD;	// LW18 
TEMP9:WORD;	// LW20 
TEMP10:WORD;	// LW22 
TEMP11:WORD;	// LW24 
TEMP12:WORD;	// LW26 
TEMP13:WORD;	// LW28 
TEMP14:WORD;	// LW30 
TEMP15:WORD;	// LW32 
TEMP16:WORD;	// LW34 
TEMP17:WORD;	// LW36 
TEMP18:WORD;	// LW38 
TEMP19:WORD;	// LW40 
TEMP20:WORD;	// LW42 
TEMP21:WORD;	// LW44 
END_VAR
BEGIN
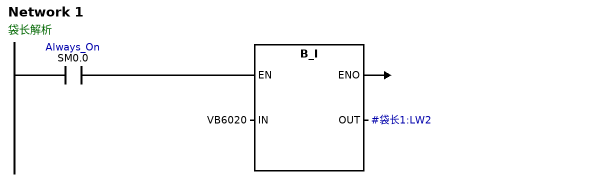
Network 1
// 袋长解析
LD     Always_On:SM0.0
BTI    VB6020, #袋长1:LW2
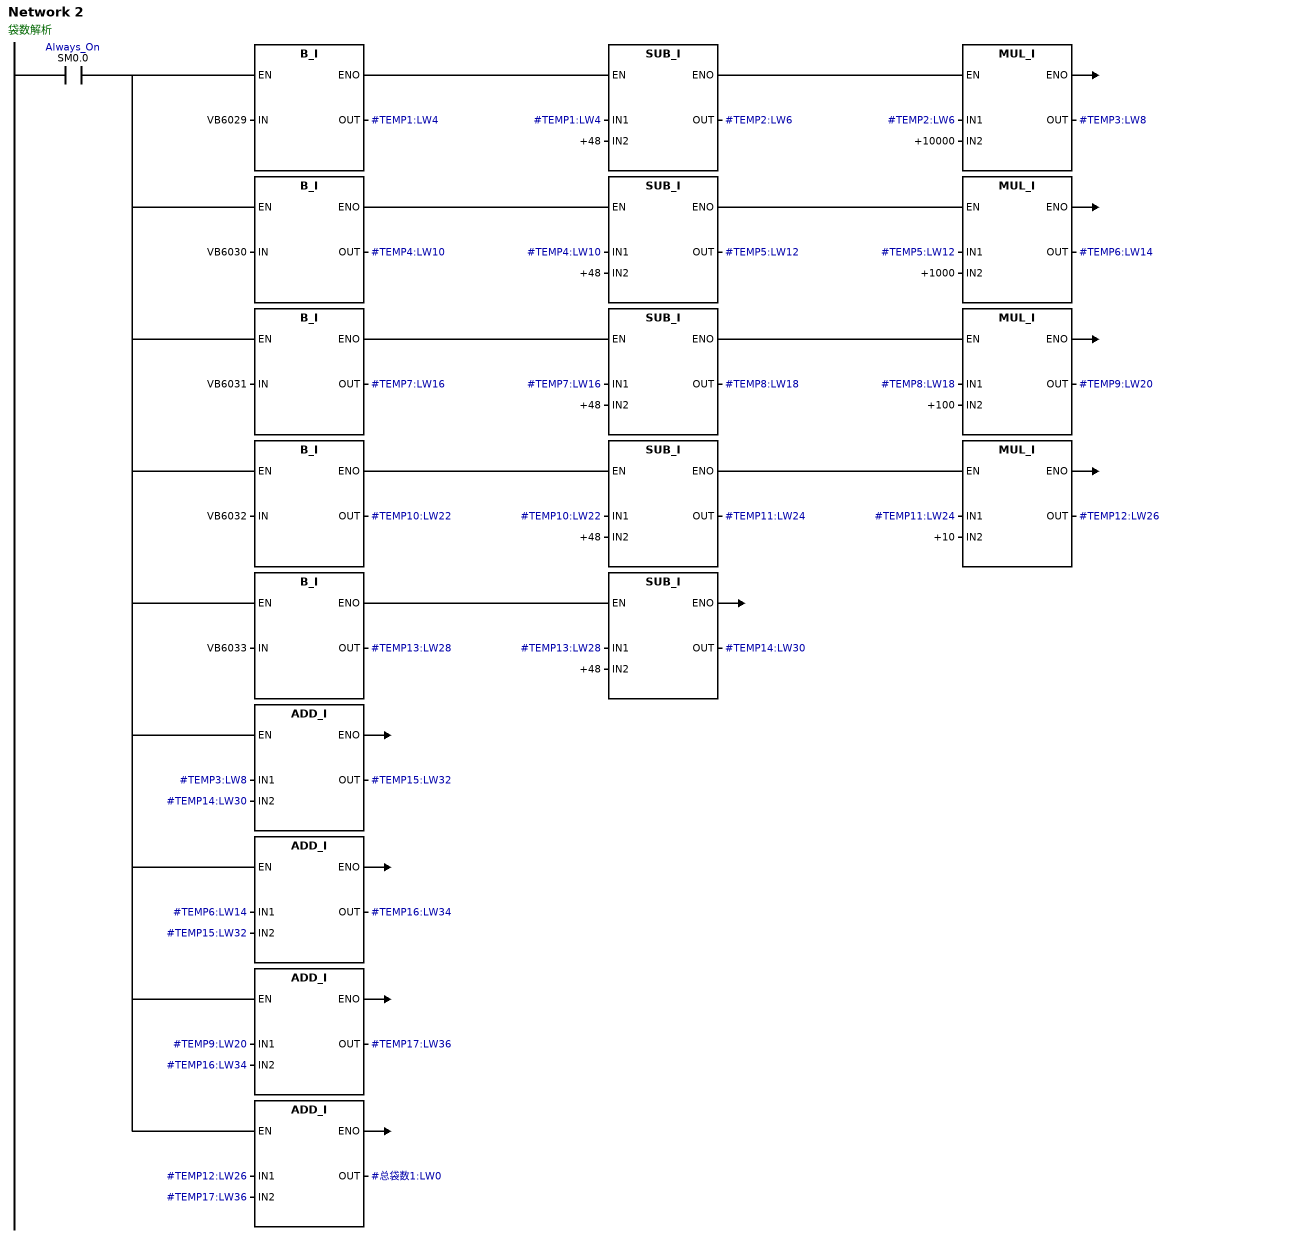
Network 2
// 袋数解析
LD     Always_On:SM0.0
LPS
BTI    VB6029, #TEMP1:LW4
AENO
MOVW   #TEMP1:LW4, #TEMP2:LW6
AENO
-I     +48, #TEMP2:LW6
AENO
MOVW   #TEMP2:LW6, #TEMP3:LW8
*I     +10000, #TEMP3:LW8
LRD
BTI    VB6030, #TEMP4:LW10
AENO
MOVW   #TEMP4:LW10, #TEMP5:LW12
AENO
-I     +48, #TEMP5:LW12
AENO
MOVW   #TEMP5:LW12, #TEMP6:LW14
*I     +1000, #TEMP6:LW14
LRD
BTI    VB6031, #TEMP7:LW16
AENO
MOVW   #TEMP7:LW16, #TEMP8:LW18
AENO
-I     +48, #TEMP8:LW18
AENO
MOVW   #TEMP8:LW18, #TEMP9:LW20
*I     +100, #TEMP9:LW20
LRD
BTI    VB6032, #TEMP10:LW22
AENO
MOVW   #TEMP10:LW22, #TEMP11:LW24
AENO
-I     +48, #TEMP11:LW24
AENO
MOVW   #TEMP11:LW24, #TEMP12:LW26
*I     +10, #TEMP12:LW26
LRD
BTI    VB6033, #TEMP13:LW28
AENO
MOVW   #TEMP13:LW28, #TEMP14:LW30
-I     +48, #TEMP14:LW30
LRD
MOVW   #TEMP3:LW8, #TEMP15:LW32
+I     #TEMP14:LW30, #TEMP15:LW32
LRD
MOVW   #TEMP6:LW14, #TEMP16:LW34
+I     #TEMP15:LW32, #TEMP16:LW34
LRD
MOVW   #TEMP9:LW20, #TEMP17:LW36
+I     #TEMP16:LW34, #TEMP17:LW36
LPP
MOVW   #TEMP12:LW26, #总袋数1:LW0
+I     #TEMP17:LW36, #总袋数1:LW0
END_SUBROUTINE_BLOCK

SUBROUTINE_BLOCK N7收:SBR27
TITLE=
VAR_OUTPUT
总袋数1:WORD;	// LW0 
袋长1:WORD;	// LW2 
END_VAR
VAR
TEMP1:WORD;	// LW4 
TEMP2:WORD;	// LW6 
TEMP3:WORD;	// LW8 
TEMP4:WORD;	// LW10 
TEMP5:WORD;	// LW12 
TEMP6:WORD;	// LW14 
TEMP7:WORD;	// LW16 
TEMP8:WORD;	// LW18 
TEMP9:WORD;	// LW20 
TEMP10:WORD;	// LW22 
TEMP11:WORD;	// LW24 
TEMP12:WORD;	// LW26 
TEMP13:WORD;	// LW28 
TEMP14:WORD;	// LW30 
TEMP15:WORD;	// LW32 
TEMP16:WORD;	// LW34 
TEMP17:WORD;	// LW36 
TEMP18:WORD;	// LW38 
TEMP19:WORD;	// LW40 
TEMP20:WORD;	// LW42 
TEMP21:WORD;	// LW44 
END_VAR
BEGIN
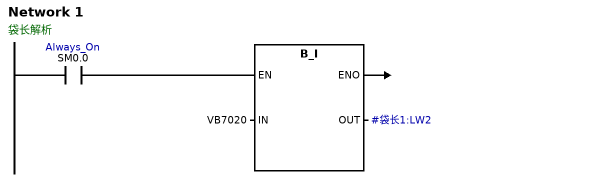
Network 1
// 袋长解析
LD     Always_On:SM0.0
BTI    VB7020, #袋长1:LW2
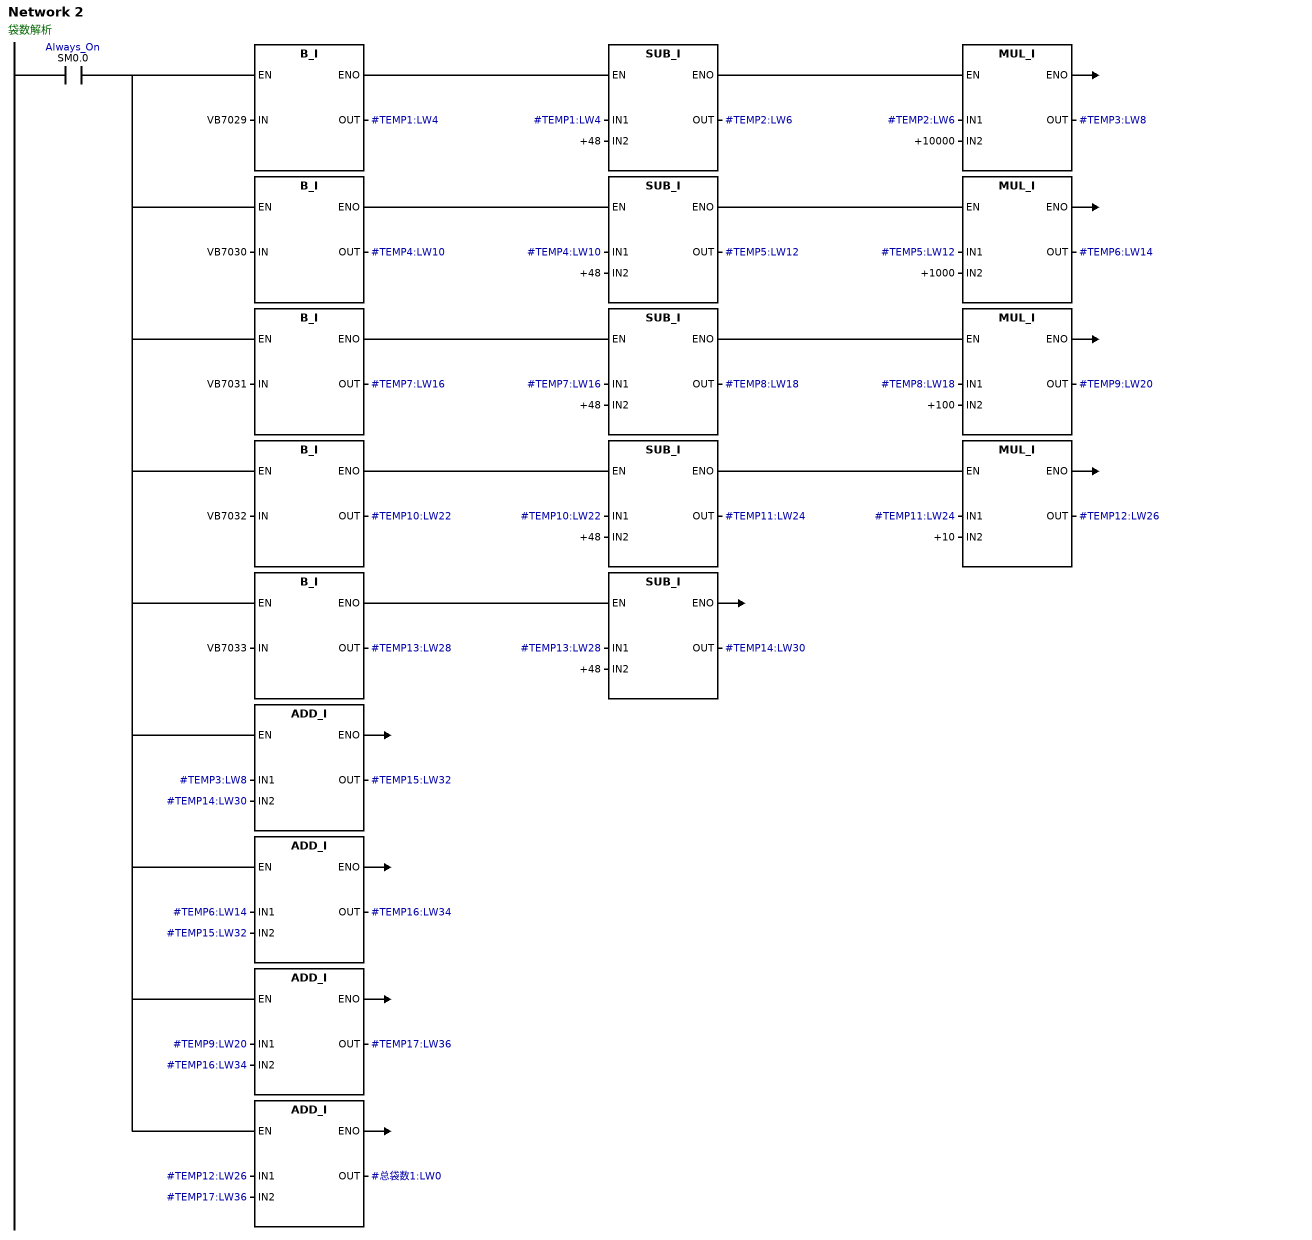
Network 2
// 袋数解析
LD     Always_On:SM0.0
LPS
BTI    VB7029, #TEMP1:LW4
AENO
MOVW   #TEMP1:LW4, #TEMP2:LW6
AENO
-I     +48, #TEMP2:LW6
AENO
MOVW   #TEMP2:LW6, #TEMP3:LW8
*I     +10000, #TEMP3:LW8
LRD
BTI    VB7030, #TEMP4:LW10
AENO
MOVW   #TEMP4:LW10, #TEMP5:LW12
AENO
-I     +48, #TEMP5:LW12
AENO
MOVW   #TEMP5:LW12, #TEMP6:LW14
*I     +1000, #TEMP6:LW14
LRD
BTI    VB7031, #TEMP7:LW16
AENO
MOVW   #TEMP7:LW16, #TEMP8:LW18
AENO
-I     +48, #TEMP8:LW18
AENO
MOVW   #TEMP8:LW18, #TEMP9:LW20
*I     +100, #TEMP9:LW20
LRD
BTI    VB7032, #TEMP10:LW22
AENO
MOVW   #TEMP10:LW22, #TEMP11:LW24
AENO
-I     +48, #TEMP11:LW24
AENO
MOVW   #TEMP11:LW24, #TEMP12:LW26
*I     +10, #TEMP12:LW26
LRD
BTI    VB7033, #TEMP13:LW28
AENO
MOVW   #TEMP13:LW28, #TEMP14:LW30
-I     +48, #TEMP14:LW30
LRD
MOVW   #TEMP3:LW8, #TEMP15:LW32
+I     #TEMP14:LW30, #TEMP15:LW32
LRD
MOVW   #TEMP6:LW14, #TEMP16:LW34
+I     #TEMP15:LW32, #TEMP16:LW34
LRD
MOVW   #TEMP9:LW20, #TEMP17:LW36
+I     #TEMP16:LW34, #TEMP17:LW36
LPP
MOVW   #TEMP12:LW26, #总袋数1:LW0
+I     #TEMP17:LW36, #总袋数1:LW0
END_SUBROUTINE_BLOCK

SUBROUTINE_BLOCK N8收:SBR28
TITLE=
VAR_OUTPUT
总袋数1:WORD;	// LW0 
袋长1:WORD;	// LW2 
END_VAR
VAR
TEMP1:WORD;	// LW4 
TEMP2:WORD;	// LW6 
TEMP3:WORD;	// LW8 
TEMP4:WORD;	// LW10 
TEMP5:WORD;	// LW12 
TEMP6:WORD;	// LW14 
TEMP7:WORD;	// LW16 
TEMP8:WORD;	// LW18 
TEMP9:WORD;	// LW20 
TEMP10:WORD;	// LW22 
TEMP11:WORD;	// LW24 
TEMP12:WORD;	// LW26 
TEMP13:WORD;	// LW28 
TEMP14:WORD;	// LW30 
TEMP15:WORD;	// LW32 
TEMP16:WORD;	// LW34 
TEMP17:WORD;	// LW36 
TEMP18:WORD;	// LW38 
TEMP19:WORD;	// LW40 
TEMP20:WORD;	// LW42 
TEMP21:WORD;	// LW44 
END_VAR
BEGIN
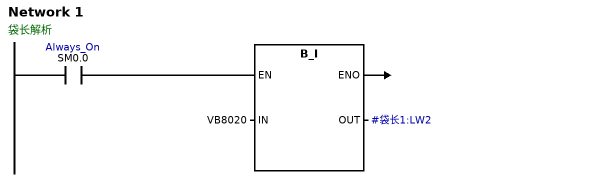
Network 1
// 袋长解析
LD     Always_On:SM0.0
BTI    VB8020, #袋长1:LW2
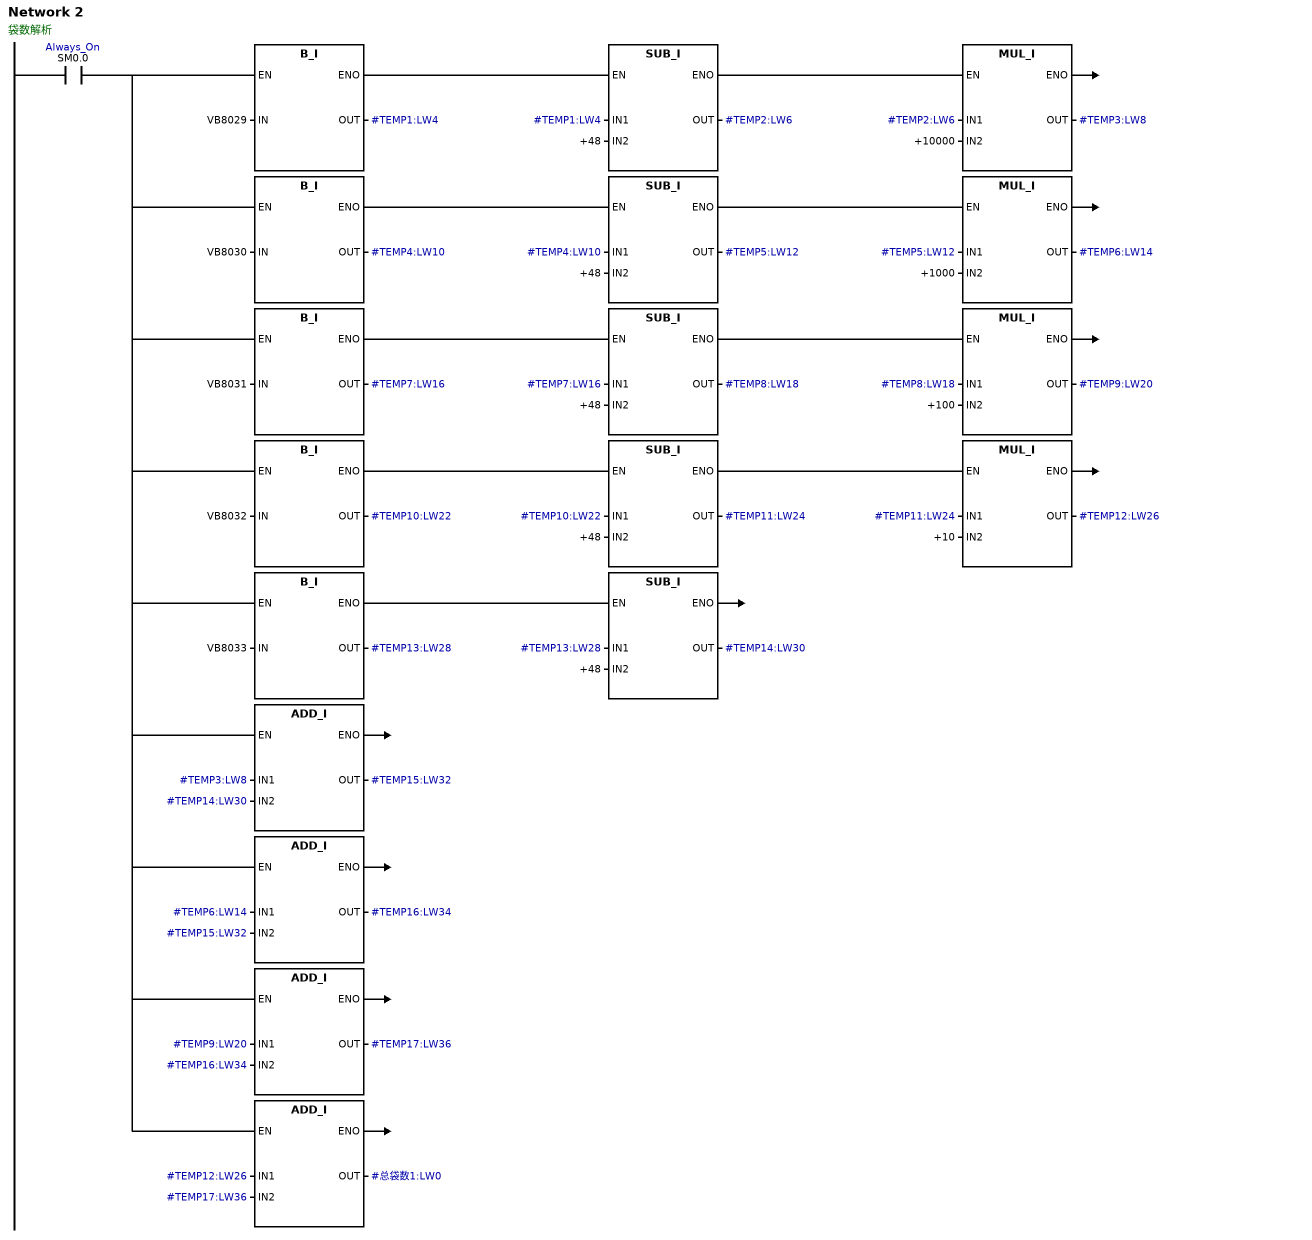
Network 2
// 袋数解析
LD     Always_On:SM0.0
LPS
BTI    VB8029, #TEMP1:LW4
AENO
MOVW   #TEMP1:LW4, #TEMP2:LW6
AENO
-I     +48, #TEMP2:LW6
AENO
MOVW   #TEMP2:LW6, #TEMP3:LW8
*I     +10000, #TEMP3:LW8
LRD
BTI    VB8030, #TEMP4:LW10
AENO
MOVW   #TEMP4:LW10, #TEMP5:LW12
AENO
-I     +48, #TEMP5:LW12
AENO
MOVW   #TEMP5:LW12, #TEMP6:LW14
*I     +1000, #TEMP6:LW14
LRD
BTI    VB8031, #TEMP7:LW16
AENO
MOVW   #TEMP7:LW16, #TEMP8:LW18
AENO
-I     +48, #TEMP8:LW18
AENO
MOVW   #TEMP8:LW18, #TEMP9:LW20
*I     +100, #TEMP9:LW20
LRD
BTI    VB8032, #TEMP10:LW22
AENO
MOVW   #TEMP10:LW22, #TEMP11:LW24
AENO
-I     +48, #TEMP11:LW24
AENO
MOVW   #TEMP11:LW24, #TEMP12:LW26
*I     +10, #TEMP12:LW26
LRD
BTI    VB8033, #TEMP13:LW28
AENO
MOVW   #TEMP13:LW28, #TEMP14:LW30
-I     +48, #TEMP14:LW30
LRD
MOVW   #TEMP3:LW8, #TEMP15:LW32
+I     #TEMP14:LW30, #TEMP15:LW32
LRD
MOVW   #TEMP6:LW14, #TEMP16:LW34
+I     #TEMP15:LW32, #TEMP16:LW34
LRD
MOVW   #TEMP9:LW20, #TEMP17:LW36
+I     #TEMP16:LW34, #TEMP17:LW36
LPP
MOVW   #TEMP12:LW26, #总袋数1:LW0
+I     #TEMP17:LW36, #总袋数1:LW0
END_SUBROUTINE_BLOCK

SUBROUTINE_BLOCK ZBKZ:SBR29
TITLE=子程序注释
BEGIN
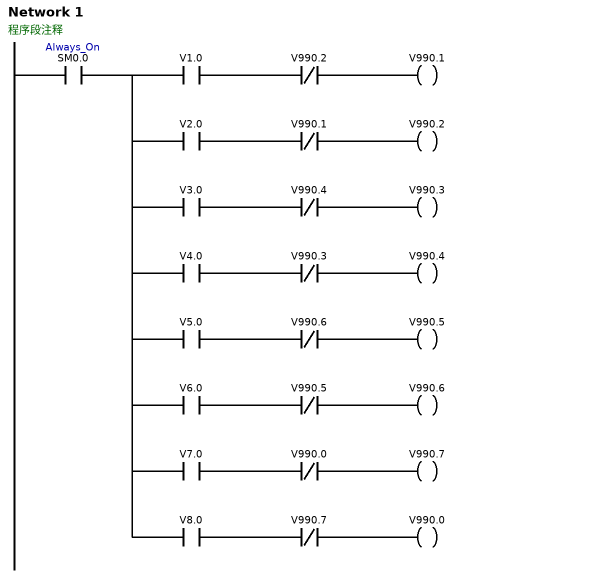
Network 1
// 程序段注释
LD     Always_On:SM0.0
LPS
A      V1.0
AN     V990.2
=      V990.1
LRD
A      V2.0
AN     V990.1
=      V990.2
LRD
A      V3.0
AN     V990.4
=      V990.3
LRD
A      V4.0
AN     V990.3
=      V990.4
LRD
A      V5.0
AN     V990.6
=      V990.5
LRD
A      V6.0
AN     V990.5
=      V990.6
LRD
A      V7.0
AN     V990.0
=      V990.7
LPP
A      V8.0
AN     V990.7
=      V990.0
